FUNCTION_BLOCK fbPPPSKlimatyzatorTroxSchoolairV
  VAR_INPUT
    sKomunikat : alSTRINGKomunikat;  (* komunikat z systemu zewnętrznego *)
    intTablicaKomunikatowRozmiar : INT;  (* rozmiar tablicy danych wysyłkowych *)
    intModbusOdczytZapisZadanieRozmiar : INT;  (* rozmiar tablicy danych modbusa *)
    xTablicaKomunikatowHold : BOOL;  (* wstrzymanie komunikacji mniej ważnych komunikatów *)
    sIdInstancji : STRING;  (* parametr ID rolety np NS02L*202IBM**** *)
    sIdAplikacji : STRING;  (* parametr ID aplikacji np SO*******ECL*000 *)
    sMnemonik : STRING;  (* mnemonik właściciela - BCB* *)
    sMACAdres : STRING;  (* MAC adres sterownika *)
    sDaneZapasowe : STRING;  (* 6 znaków zapasu *)
    tCzasOpoznieniaRestartu : TIME;  (* czas opóźnienia po którym zaczynają być raportowane wartości *)
    tCzasOpoznieniaAlarmu : TIME := TIME#1m0s0ms;  (* czas opóźnienia po którym zaczynają być raportowane wartości *)
    bAdres : BYTE;
    tMinimalnyCzasRaportowania : TIME;
    tMaksymalnyCzasRaportowania : TIME;
    xAutonomizacja : BOOL;
    xAutonomizacjaSztuczna : BOOL;
  END_VAR
  VAR_IN_OUT
    arModbusOdczytCykliczny : ARRAY[1..5000] OF typModbusOdczytCykliczny;
    arModbusStatusKomunikacji : ARRAY[1..256] OF INT;
    arModbusOdczytZapisZadanie : ARRAY[1..1000] OF typModbusOdczytZapisZadanie;
    intModbusOdczytZapisZadanieZnacznikZapisu : INT;
    arTablicaKomunikatow : alARRAYTablicaKomunikatow;
    intTablicaKomunikatowZnacznikZapisu : INT;
  END_VAR
  VAR
    xPoInicjalizacji : BOOL := FALSE;  (* Inicjalizacja *)
    fbInicjalizacyjnyTimer : TON;
    tCzasInicjalizacji : TIME := TIME#30s0ms;
    xPierwszySkan : BOOL := TRUE;  (* Definicje zmiennych do odczytu wartości z modbusa *)
    intPetlaPierwszySkan : INT := 1;
    sDane : alSTRINGKomunikat;  (* Definicje do komunikacji z IZE *)
    sWyslanyKomunikat : alSTRINGKomunikat;
    sWyslanyKomunikatDummy : alSTRINGKomunikat;
    xZadanieRaportu : BOOL;
    sKomunikatPamiec : alSTRINGKomunikat;
    intPetla : INT;
    arErrorStan : ARRAY[0..10] OF INT;  (* tablica przechowująca statusy alarmowe *)
    arErrorKlasa : ARRAY[0..10] OF INT;  (* tablica przechowująca klasy danych alarmów *)
    xRaport : BOOL := FALSE;
    sTempWartoscAtrybutu : STRING;
    xOverFlow : BOOL;
    fbTimerBrakuKomunikacji : TON;  (* Kontrola komunikacji urządzenia *)
    xBrakKomunikacjiPLC : BOOL;
    xBrakKomunikacjiIZE : BOOL;
    intBlokadaWykonywaniaRozkazow : INT;  (* Parametry *)
    intBlokadaWykonywaniaRozkazowZaraportowana : INT;
    wTrybPracy : WORD;  (* 255 = Nul, 0 = Occupied, 1 = Unoccupied, 2 = Boost, 3 = Standby *)
    rTrybPracy : REAL;
    rTrybPracyZaraportowana : REAL;
    wPredkoscWentylatora : WORD;  (* High-Byte: Value, Low-Byte: 0 Auto, 1 Hand *)
    rPredkoscWentylatora : REAL;
    rPredkoscWentylatoraZaraportowana : REAL;  (* 40 = Level 1, 80 = Level 2, 120 = Level 3, 160 = Level 4, 200 = Level 5 *)
    fbPredkoscWentylatora : fbFiltrWartoscAnalogowa;
    wTrybOperacji : WORD;  (* 255 = HVAC_NUL, 0 = HVAC_AUTO, 1 = HVAC_HEAT, 2 = HVAC_MRNG_WRMUP, 3 = HVAC_COOL, 4 = HVAC_NIGHT_PURGE, 5 = HVAC_PRE_COOL, 6 = HVAC_OFF *)
    rTrybOperacji : REAL;  (* 7 = HVAC_TEST, 8 = HVAC_EMERG_HEAT, 9 = HVAC_FAN_ONLY, 10 = HVAC_FREE_COOL, 12 = HVAC_MAXHEAT, 13 = HVAC_ECONOMY, 14 = HVAC_DEHUMID *)
    rTrybOperacjiZaraportowana : REAL;
    wTemperaturaReferencyjna : WORD;  (* Unit 0.01°C *)
    rTemperaturaReferencyjna : REAL;
    rTemperaturaReferencyjnaZaraportowana : REAL;
    wTemperaturaRzeczywista : WORD;  (* Unit 0.01°C *)
    rTemperaturaRzeczywista : REAL;
    rTemperaturaRzeczywistaZaraportowana : REAL;
    fbTemperaturaRzeczywista : fbFiltrWartoscAnalogowa;
    rTemperaturaRzeczywistaPamiec : REAL;
    xBrakZmianyTemperatury : BOOL;
    fbBrakZmianyTemperaturyTimer : TON;
    xBladBrakZmianyTemperatury : BOOL;
  END_VAR

            (*			
Autor:					Artur Wyszomirski, 2019-03-08 
Prawa majątkowe: 		Solwena Sp. z o.o., 
Aktualizacje:			2019-05-16-AWy: Modyfikacja warunku na raportowanie. Dopisane: AND arModbusStatusKomunikacji[bAdres] = enumModbusStatus.KomunikacjaPrawidlowa AND xPoInicjalizacji 
						
Opis:					fb służy do komunikacji z klimatyzatorem Trox Schoolair V
				
*)


// Inicjalizacja sterownika
fbInicjalizacyjnyTimer(IN := (NOT xPoInicjalizacji AND arModbusStatusKomunikacji[bAdres] = enumModbusStatus.KomunikacjaPrawidlowa) , PT := tCzasOpoznieniaRestartu);
IF fbInicjalizacyjnyTimer.Q THEN
	rTrybPracyZaraportowana := rTrybPracy;
	rPredkoscWentylatoraZaraportowana := rPredkoscWentylatora;
	rTrybOperacji := rTrybOperacjiZaraportowana;
	rTemperaturaReferencyjnaZaraportowana := rTemperaturaReferencyjna;
	rTemperaturaRzeczywistaZaraportowana := rTemperaturaRzeczywista;
	xPoInicjalizacji := TRUE;
END_IF
//

IF xAutonomizacjaSztuczna = TRUE THEN
	xAutonomizacja := TRUE;
END_IF 

// Kontrola komunikacji
fbTimerBrakuKomunikacji(IN := arModbusStatusKomunikacji[bAdres] = enumModbusStatus.BrakKomunikacji, PT := T#60S);
IF fbTimerBrakuKomunikacji.Q THEN
	xBrakKomunikacjiPLC := TRUE;
ELSE
	xBrakKomunikacjiPLC := FALSE;
END_IF

IF xAutonomizacja THEN
	xBrakKomunikacjiIZE := TRUE;
ELSE
	xBrakKomunikacjiIZE := FALSE;
END_IF
//

IF xPierwszySkan THEN
	xPierwszySkan := FALSE;
	WHILE arModbusOdczytCykliczny[intPetlaPierwszySkan].bAdresUrzadzenia <> 0 DO
		intPetlaPierwszySkan := intPetlaPierwszySkan + 1;
	END_WHILE

	arModbusOdczytCykliczny[intPetlaPierwszySkan].bAdresUrzadzenia := bAdres;
	arModbusOdczytCykliczny[intPetlaPierwszySkan].bFunkcja := TO_BYTE(enumModbusKodyFunkcji.OdczytNRejestrowWejsciowych);
	arModbusOdczytCykliczny[intPetlaPierwszySkan].uiAdresRejestru := 17;
	arModbusOdczytCykliczny[intPetlaPierwszySkan].ltCzestotliwosc := TIME_TO_LTIME(tMinimalnyCzasRaportowania);
	arModbusOdczytCykliczny[intPetlaPierwszySkan].pZmiennaReferencyjna := ADR(wTrybPracy);
	intPetlaPierwszySkan := intPetlaPierwszySkan + 1;	
	
	arModbusOdczytCykliczny[intPetlaPierwszySkan].bAdresUrzadzenia := bAdres;
	arModbusOdczytCykliczny[intPetlaPierwszySkan].bFunkcja := TO_BYTE(enumModbusKodyFunkcji.OdczytNRejestrowWejsciowych);
	arModbusOdczytCykliczny[intPetlaPierwszySkan].uiAdresRejestru := 19;
	arModbusOdczytCykliczny[intPetlaPierwszySkan].ltCzestotliwosc := TIME_TO_LTIME(tMinimalnyCzasRaportowania);
	arModbusOdczytCykliczny[intPetlaPierwszySkan].pZmiennaReferencyjna := ADR(wTemperaturaReferencyjna);
	intPetlaPierwszySkan := intPetlaPierwszySkan + 1;		
	
	arModbusOdczytCykliczny[intPetlaPierwszySkan].bAdresUrzadzenia := bAdres;
	arModbusOdczytCykliczny[intPetlaPierwszySkan].bFunkcja := TO_BYTE(enumModbusKodyFunkcji.OdczytNRejestrowWejsciowych);
	arModbusOdczytCykliczny[intPetlaPierwszySkan].uiAdresRejestru := 21;
	arModbusOdczytCykliczny[intPetlaPierwszySkan].ltCzestotliwosc := TIME_TO_LTIME(tMinimalnyCzasRaportowania);
	arModbusOdczytCykliczny[intPetlaPierwszySkan].pZmiennaReferencyjna := ADR(wPredkoscWentylatora);
	intPetlaPierwszySkan := intPetlaPierwszySkan + 1;

	arModbusOdczytCykliczny[intPetlaPierwszySkan].bAdresUrzadzenia := bAdres;
	arModbusOdczytCykliczny[intPetlaPierwszySkan].bFunkcja := TO_BYTE(enumModbusKodyFunkcji.OdczytNRejestrowWejsciowych);
	arModbusOdczytCykliczny[intPetlaPierwszySkan].uiAdresRejestru := 22;
	arModbusOdczytCykliczny[intPetlaPierwszySkan].ltCzestotliwosc := TIME_TO_LTIME(tMinimalnyCzasRaportowania);
	arModbusOdczytCykliczny[intPetlaPierwszySkan].pZmiennaReferencyjna := ADR(wTrybOperacji);
	intPetlaPierwszySkan := intPetlaPierwszySkan + 1;

	arModbusOdczytCykliczny[intPetlaPierwszySkan].bAdresUrzadzenia := bAdres;
	arModbusOdczytCykliczny[intPetlaPierwszySkan].bFunkcja := TO_BYTE(enumModbusKodyFunkcji.OdczytNRejestrowWejsciowych);
	arModbusOdczytCykliczny[intPetlaPierwszySkan].uiAdresRejestru := 25;
	arModbusOdczytCykliczny[intPetlaPierwszySkan].ltCzestotliwosc := TIME_TO_LTIME(tMinimalnyCzasRaportowania);
	arModbusOdczytCykliczny[intPetlaPierwszySkan].pZmiennaReferencyjna := ADR(wTemperaturaRzeczywista);
	intPetlaPierwszySkan := intPetlaPierwszySkan + 1;							
END_IF

// Przeliczenie zmiennych
rTrybPracy := WORD_TO_REAL(wTrybPracy);
rPredkoscWentylatora := WORD_TO_REAL(SHR((wPredkoscWentylatora AND 16#FF00),8));
rTrybOperacji := WORD_TO_REAL(wTrybOperacji);
rTemperaturaReferencyjna := WORD_TO_REAL(wTemperaturaReferencyjna)*0.01 + 273.15;

fbTemperaturaRzeczywista(	rWartoscWejsciowa := WORD_TO_REAL(wTemperaturaRzeczywista),
							rDeadband := 0.5,
							tCzasMinimalny := tMinimalnyCzasRaportowania,
							tCzasMaksymalny := tMaksymalnyCzasRaportowania,
							rWynikMnoznik := 0.01,
							rWynikOffset := 273.15,
							rWartoscWejsciowaZaraportowana := rTemperaturaRzeczywistaZaraportowana,
							rWartoscWyjsciowa => rTemperaturaRzeczywista);
//					
						
						
// Obsluga komunikatu przychodzacego z IZE
IF sKomunikat <> sKomunikatPamiec AND xPoInicjalizacji THEN
	sKomunikatPamiec := sKomunikat;
	IF fnIDOdbiorcyMatch(sKomunikat , sIdInstancji) THEN
		sDane := '';
		// Rozkaz typu C
		IF fnKomunikatTyp(sKomunikat) = 'C' AND NOT xAutonomizacja THEN
			IF fnKomunikatDaneSzukajWartosci(sKomunikat,'BLOK=') = '0' THEN
				IF intBlokadaWykonywaniaRozkazow = 1 THEN
					intBlokadaWykonywaniaRozkazow := 0;
					xRaport := TRUE;
					ELSE	
					IF sDane <> '' THEN
					sDane := CONCAT(sDane , ';');
					END_IF
					sDane := CONCAT(sDane , 'BLOK=0');
				END_IF
			END_IF
			IF fnKomunikatDaneSzukajWartosci(sKomunikat,'BLOK=') = '1' THEN
				IF intBlokadaWykonywaniaRozkazow = 0 THEN
					intBlokadaWykonywaniaRozkazow := 1;
					xRaport := TRUE;
					ELSE
					IF sDane <> '' THEN
					sDane := CONCAT(sDane , ';');
					END_IF					
					sDane := CONCAT(sDane , 'BLOK=1');
				END_IF
			END_IF
		END_IF
				
		// Zapytanie typu Q
		IF fnKomunikatTyp(sKomunikat) = 'Q' AND arModbusStatusKomunikacji[bAdres] = enumModbusStatus.KomunikacjaPrawidlowa THEN
			IF fnKomunikatDaneSzukajWartosci(sKomunikat , 'BLOK=') = '?' OR fnKomunikatDaneSzukajWartosci(sKomunikat , 'ALL=') = '?' THEN
				fnKomunikatDaneDodaj_xOverFlow(sDane := sDane , sAtrybut := 'BLOK=' , sWartosc := INT_TO_STRING(intBlokadaWykonywaniaRozkazow) , xOverFlow := xOverFlow);	
				IF xOverFlow = TRUE THEN
					fnZapiszKomunikat(	sCalyKomunikat := '' ,
								sTypKomunikatu := 'A' ,
								sMnemonik := sMnemonik ,
								sMACAdres := sMACAdres ,
								sIDNadawcy := sIdInstancji ,
								sIDOdbiorcy := sIdAplikacji ,
								sDaneZapasowe := sDaneZapasowe ,
								sDane := sDane ,
								arTablicaKomunikatow := arTablicaKomunikatow ,
								intTablicaKomunikatowZnacznikZapisu := intTablicaKomunikatowZnacznikZapisu ,
								intTablicaKomunikatowRozmiar := intTablicaKomunikatowRozmiar ,
								sWyslanyKomunikat := sWyslanyKomunikatDummy);
					sDane := '';
				END_IF
			END_IF
			IF fnKomunikatDaneSzukajWartosci(sKomunikat , 'TRYBPRACY=') = '?' OR fnKomunikatDaneSzukajWartosci(sKomunikat , 'ALL=') = '?' THEN
				fnKomunikatDaneDodaj_xOverFlow(sDane := sDane , sAtrybut := 'TRYBPRACY=' , sWartosc := REAL_TO_STRING(rTrybPracy) , xOverFlow := xOverFlow);	
				IF xOverFlow = TRUE THEN
					fnZapiszKomunikat(	sCalyKomunikat := '' ,
								sTypKomunikatu := 'A' ,
								sMnemonik := sMnemonik ,
								sMACAdres := sMACAdres ,
								sIDNadawcy := sIdInstancji ,
								sIDOdbiorcy := sIdAplikacji ,
								sDaneZapasowe := sDaneZapasowe ,
								sDane := sDane ,
								arTablicaKomunikatow := arTablicaKomunikatow ,
								intTablicaKomunikatowZnacznikZapisu := intTablicaKomunikatowZnacznikZapisu ,
								intTablicaKomunikatowRozmiar := intTablicaKomunikatowRozmiar ,
								sWyslanyKomunikat := sWyslanyKomunikatDummy);
					sDane := '';
				END_IF
			END_IF		
			IF fnKomunikatDaneSzukajWartosci(sKomunikat , 'PREDKOSCWENT=') = '?' OR fnKomunikatDaneSzukajWartosci(sKomunikat , 'ALL=') = '?' THEN
				fnKomunikatDaneDodaj_xOverFlow(sDane := sDane , sAtrybut := 'PREDKOSCWENT=' , sWartosc := REAL_TO_STRING(rPredkoscWentylatora) , xOverFlow := xOverFlow);	
				IF xOverFlow = TRUE THEN
					fnZapiszKomunikat(	sCalyKomunikat := '' ,
								sTypKomunikatu := 'A' ,
								sMnemonik := sMnemonik ,
								sMACAdres := sMACAdres ,
								sIDNadawcy := sIdInstancji ,
								sIDOdbiorcy := sIdAplikacji ,
								sDaneZapasowe := sDaneZapasowe ,
								sDane := sDane ,
								arTablicaKomunikatow := arTablicaKomunikatow ,
								intTablicaKomunikatowZnacznikZapisu := intTablicaKomunikatowZnacznikZapisu ,
								intTablicaKomunikatowRozmiar := intTablicaKomunikatowRozmiar ,
								sWyslanyKomunikat := sWyslanyKomunikatDummy);
					sDane := '';
				END_IF
			END_IF		
			IF fnKomunikatDaneSzukajWartosci(sKomunikat , 'TEMPREF=') = '?' OR fnKomunikatDaneSzukajWartosci(sKomunikat , 'ALL=') = '?' THEN
				fnKomunikatDaneDodaj_xOverFlow(sDane := sDane , sAtrybut := 'TEMPREF=' , sWartosc := REAL_TO_STRING(rTemperaturaReferencyjna) , xOverFlow := xOverFlow);	
				IF xOverFlow = TRUE THEN
					fnZapiszKomunikat(	sCalyKomunikat := '' ,
								sTypKomunikatu := 'A' ,
								sMnemonik := sMnemonik ,
								sMACAdres := sMACAdres ,
								sIDNadawcy := sIdInstancji ,
								sIDOdbiorcy := sIdAplikacji ,
								sDaneZapasowe := sDaneZapasowe ,
								sDane := sDane ,
								arTablicaKomunikatow := arTablicaKomunikatow ,
								intTablicaKomunikatowZnacznikZapisu := intTablicaKomunikatowZnacznikZapisu ,
								intTablicaKomunikatowRozmiar := intTablicaKomunikatowRozmiar ,
								sWyslanyKomunikat := sWyslanyKomunikatDummy);
					sDane := '';
				END_IF
			END_IF		
			IF fnKomunikatDaneSzukajWartosci(sKomunikat , 'TEMPRZECZ=') = '?' OR fnKomunikatDaneSzukajWartosci(sKomunikat , 'ALL=') = '?' THEN
				fnKomunikatDaneDodaj_xOverFlow(sDane := sDane , sAtrybut := 'TEMPRZECZ=' , sWartosc := REAL_TO_STRING(rTemperaturaRzeczywista) , xOverFlow := xOverFlow);	
				IF xOverFlow = TRUE THEN
					fnZapiszKomunikat(	sCalyKomunikat := '' ,
								sTypKomunikatu := 'A' ,
								sMnemonik := sMnemonik ,
								sMACAdres := sMACAdres ,
								sIDNadawcy := sIdInstancji ,
								sIDOdbiorcy := sIdAplikacji ,
								sDaneZapasowe := sDaneZapasowe ,
								sDane := sDane ,
								arTablicaKomunikatow := arTablicaKomunikatow ,
								intTablicaKomunikatowZnacznikZapisu := intTablicaKomunikatowZnacznikZapisu ,
								intTablicaKomunikatowRozmiar := intTablicaKomunikatowRozmiar ,
								sWyslanyKomunikat := sWyslanyKomunikatDummy);
					sDane := '';
				END_IF
			END_IF		
			IF fnKomunikatDaneSzukajWartosci(sKomunikat , 'TRYBOP=') = '?' OR fnKomunikatDaneSzukajWartosci(sKomunikat , 'ALL=') = '?' THEN
				fnKomunikatDaneDodaj_xOverFlow(sDane := sDane , sAtrybut := 'TRYBOP=' , sWartosc := REAL_TO_STRING(rTrybOperacji) , xOverFlow := xOverFlow);	
				IF xOverFlow = TRUE THEN
					fnZapiszKomunikat(	sCalyKomunikat := '' ,
								sTypKomunikatu := 'A' ,
								sMnemonik := sMnemonik ,
								sMACAdres := sMACAdres ,
								sIDNadawcy := sIdInstancji ,
								sIDOdbiorcy := sIdAplikacji ,
								sDaneZapasowe := sDaneZapasowe ,
								sDane := sDane ,
								arTablicaKomunikatow := arTablicaKomunikatow ,
								intTablicaKomunikatowZnacznikZapisu := intTablicaKomunikatowZnacznikZapisu ,
								intTablicaKomunikatowRozmiar := intTablicaKomunikatowRozmiar ,
								sWyslanyKomunikat := sWyslanyKomunikatDummy);
					sDane := '';
				END_IF
			END_IF		
			// Pytanie o stany alarmów
			IF fnKomunikatDaneSzukajWartosci(sKomunikat , 'ALARM=') = '?' OR fnKomunikatDaneSzukajWartosci(sKomunikat , 'ALL=') = '?' THEN
				FOR intPetla := 1 TO 10 BY 1 DO
					// Raportowanie typu E (stanów alarmów) na zapytanie typu Q
					IF arErrorStan[intPetla] <> enumAlarmWartosc.StanNieznany THEN
						fnZapiszKomunikat(	sCalyKomunikat := '' ,
											sTypKomunikatu := 'E' ,
											sMnemonik := sMnemonik ,
											sMACAdres := sMACAdres ,
											sIDNadawcy := sIdInstancji ,
											sIDOdbiorcy := sIdAplikacji ,
											sDaneZapasowe := sDaneZapasowe ,
											sDane := fnKomunikatDaneErrorRetry(xAktywny := arErrorStan[intPetla] = enumAlarmWartosc.StanAlarmowy , intKlasa := arErrorKlasa[intPetla] , intNumer := intPetla),
											arTablicaKomunikatow := arTablicaKomunikatow ,
											intTablicaKomunikatowZnacznikZapisu := intTablicaKomunikatowZnacznikZapisu ,
											intTablicaKomunikatowRozmiar := intTablicaKomunikatowRozmiar ,
											sWyslanyKomunikat := sWyslanyKomunikatDummy);
					END_IF
				END_FOR
			END_IF
		END_IF		
		// Raportowanie typu A na zapytanie Q
		IF sDane <> '' THEN
			fnZapiszKomunikat(	sCalyKomunikat := '' ,
								sTypKomunikatu := 'A' ,
								sMnemonik := sMnemonik ,
								sMACAdres := sMACAdres ,
								sIDNadawcy := sIdInstancji ,
								sIDOdbiorcy := sIdAplikacji ,
								sDaneZapasowe := sDaneZapasowe ,
								sDane := sDane ,
								arTablicaKomunikatow := arTablicaKomunikatow ,
								intTablicaKomunikatowZnacznikZapisu := intTablicaKomunikatowZnacznikZapisu ,
								intTablicaKomunikatowRozmiar := intTablicaKomunikatowRozmiar ,
								sWyslanyKomunikat := sWyslanyKomunikatDummy);
		END_IF
	END_IF
END_IF

// Raportowanie typu M do IZE wartosci odczytanych z Modbusa	
IF 	(intBlokadaWykonywaniaRozkazow <> intBlokadaWykonywaniaRozkazowZaraportowana OR rTrybPracy <> rTrybPracyZaraportowana OR rPredkoscWentylatora <> rPredkoscWentylatoraZaraportowana OR
	rTemperaturaReferencyjna <> rTemperaturaReferencyjnaZaraportowana OR rTemperaturaRzeczywista <> rTemperaturaRzeczywistaZaraportowana OR rTrybOperacji <> rTrybOperacjiZaraportowana) AND 
	arModbusStatusKomunikacji[bAdres] = enumModbusStatus.KomunikacjaPrawidlowa AND xPoInicjalizacji THEN
	xRaport := TRUE;
END_IF

IF xRaport THEN
	sDane := '';
	xRaport := FALSE;
	IF intBlokadaWykonywaniaRozkazow <> intBlokadaWykonywaniaRozkazowZaraportowana THEN 
		intBlokadaWykonywaniaRozkazowZaraportowana := intBlokadaWykonywaniaRozkazow;
		fnKomunikatDaneDodaj_xOverFlow(sDane := sDane , sAtrybut := 'BLOK=' , sWartosc := INT_TO_STRING(intBlokadaWykonywaniaRozkazow) , xOverFlow := xOverFlow);	
	END_IF	
	IF xOverFlow = TRUE THEN
		fnZapiszKomunikat(	sCalyKomunikat := '' ,
					sTypKomunikatu := 'M' ,
					sMnemonik := sMnemonik ,
					sMACAdres := sMACAdres ,
					sIDNadawcy := sIdInstancji ,
					sIDOdbiorcy := sIdAplikacji ,
					sDaneZapasowe := sDaneZapasowe ,
					sDane := sDane ,
					arTablicaKomunikatow := arTablicaKomunikatow ,
					intTablicaKomunikatowZnacznikZapisu := intTablicaKomunikatowZnacznikZapisu ,
					intTablicaKomunikatowRozmiar := intTablicaKomunikatowRozmiar ,
					sWyslanyKomunikat := sWyslanyKomunikatDummy);
		sDane := '';
	END_IF
	// Tryb pracy
	IF rTrybPracy <> rTrybPracyZaraportowana THEN
		rTrybPracyZaraportowana := rTrybPracy;
		fnKomunikatDaneDodaj_xOverFlow(sDane := sDane , sAtrybut := 'TRYBPRACY=' , sWartosc := REAL_TO_STRING(rTrybPracy) , xOverFlow := xOverFlow);	
		IF xOverFlow = TRUE THEN
			fnZapiszKomunikat(	sCalyKomunikat := '' ,
						sTypKomunikatu := 'M' ,
						sMnemonik := sMnemonik ,
						sMACAdres := sMACAdres ,
						sIDNadawcy := sIdInstancji ,
						sIDOdbiorcy := sIdAplikacji ,
						sDaneZapasowe := sDaneZapasowe ,
						sDane := sDane ,
						arTablicaKomunikatow := arTablicaKomunikatow ,
						intTablicaKomunikatowZnacznikZapisu := intTablicaKomunikatowZnacznikZapisu ,
						intTablicaKomunikatowRozmiar := intTablicaKomunikatowRozmiar ,
						sWyslanyKomunikat := sWyslanyKomunikatDummy);
			sDane := '';
		END_IF	
	END_IF
	// Prędkość wentylatora
	IF rPredkoscWentylatora <> rPredkoscWentylatoraZaraportowana THEN
		rPredkoscWentylatoraZaraportowana := rPredkoscWentylatora;
		fnKomunikatDaneDodaj_xOverFlow(sDane := sDane , sAtrybut := 'PREDKOSCWENT=' , sWartosc := REAL_TO_STRING(rPredkoscWentylatora) , xOverFlow := xOverFlow);	
		IF xOverFlow = TRUE THEN
			fnZapiszKomunikat(	sCalyKomunikat := '' ,
						sTypKomunikatu := 'M' ,
						sMnemonik := sMnemonik ,
						sMACAdres := sMACAdres ,
						sIDNadawcy := sIdInstancji ,
						sIDOdbiorcy := sIdAplikacji ,
						sDaneZapasowe := sDaneZapasowe ,
						sDane := sDane ,
						arTablicaKomunikatow := arTablicaKomunikatow ,
						intTablicaKomunikatowZnacznikZapisu := intTablicaKomunikatowZnacznikZapisu ,
						intTablicaKomunikatowRozmiar := intTablicaKomunikatowRozmiar ,
						sWyslanyKomunikat := sWyslanyKomunikatDummy);
			sDane := '';
		END_IF	
	END_IF
	// Temperatura referencyjna
	IF rTemperaturaReferencyjna <> rTemperaturaReferencyjnaZaraportowana THEN
		rTemperaturaReferencyjnaZaraportowana := rTemperaturaReferencyjna;
		fnKomunikatDaneDodaj_xOverFlow(sDane := sDane , sAtrybut := 'TEMPREF=' , sWartosc := REAL_TO_STRING(rTemperaturaReferencyjna) , xOverFlow := xOverFlow);	
		IF xOverFlow = TRUE THEN
			fnZapiszKomunikat(	sCalyKomunikat := '' ,
						sTypKomunikatu := 'M' ,
						sMnemonik := sMnemonik ,
						sMACAdres := sMACAdres ,
						sIDNadawcy := sIdInstancji ,
						sIDOdbiorcy := sIdAplikacji ,
						sDaneZapasowe := sDaneZapasowe ,
						sDane := sDane ,
						arTablicaKomunikatow := arTablicaKomunikatow ,
						intTablicaKomunikatowZnacznikZapisu := intTablicaKomunikatowZnacznikZapisu ,
						intTablicaKomunikatowRozmiar := intTablicaKomunikatowRozmiar ,
						sWyslanyKomunikat := sWyslanyKomunikatDummy);
			sDane := '';
		END_IF	
	END_IF
	// Temperatura rzeczywista
	IF rTemperaturaRzeczywista <> rTemperaturaRzeczywistaZaraportowana THEN
		rTemperaturaRzeczywistaZaraportowana := rTemperaturaRzeczywista;
		fnKomunikatDaneDodaj_xOverFlow(sDane := sDane , sAtrybut := 'TEMPRZECZ=' , sWartosc := REAL_TO_STRING(rTemperaturaRzeczywista) , xOverFlow := xOverFlow);	
		IF xOverFlow = TRUE THEN
			fnZapiszKomunikat(	sCalyKomunikat := '' ,
						sTypKomunikatu := 'M' ,
						sMnemonik := sMnemonik ,
						sMACAdres := sMACAdres ,
						sIDNadawcy := sIdInstancji ,
						sIDOdbiorcy := sIdAplikacji ,
						sDaneZapasowe := sDaneZapasowe ,
						sDane := sDane ,
						arTablicaKomunikatow := arTablicaKomunikatow ,
						intTablicaKomunikatowZnacznikZapisu := intTablicaKomunikatowZnacznikZapisu ,
						intTablicaKomunikatowRozmiar := intTablicaKomunikatowRozmiar ,
						sWyslanyKomunikat := sWyslanyKomunikatDummy);
			sDane := '';
		END_IF	
	END_IF
	// Temperatura referencyjna trybu manulnego
	IF rTrybOperacji <> rTrybOperacjiZaraportowana THEN
		rTrybOperacjiZaraportowana := rTrybOperacji;
		fnKomunikatDaneDodaj_xOverFlow(sDane := sDane , sAtrybut := 'TRYBOP=' , sWartosc := REAL_TO_STRING(rTrybOperacji) , xOverFlow := xOverFlow);	
		IF xOverFlow = TRUE THEN
			fnZapiszKomunikat(	sCalyKomunikat := '' ,
						sTypKomunikatu := 'M' ,
						sMnemonik := sMnemonik ,
						sMACAdres := sMACAdres ,
						sIDNadawcy := sIdInstancji ,
						sIDOdbiorcy := sIdAplikacji ,
						sDaneZapasowe := sDaneZapasowe ,
						sDane := sDane ,
						arTablicaKomunikatow := arTablicaKomunikatow ,
						intTablicaKomunikatowZnacznikZapisu := intTablicaKomunikatowZnacznikZapisu ,
						intTablicaKomunikatowRozmiar := intTablicaKomunikatowRozmiar ,
						sWyslanyKomunikat := sWyslanyKomunikatDummy);
			sDane := '';
		END_IF	
	END_IF
	IF sDane <> '' AND xPoInicjalizacji THEN
	fnZapiszKomunikat(	sCalyKomunikat := '' ,
						sTypKomunikatu := 'M' ,
						sMnemonik := sMnemonik ,
						sMACAdres := sMACAdres ,
						sIDNadawcy := sIdInstancji ,
						sIDOdbiorcy := sIdAplikacji ,
						sDaneZapasowe := sDaneZapasowe ,
						sDane := sDane ,
						arTablicaKomunikatow := arTablicaKomunikatow ,
						intTablicaKomunikatowZnacznikZapisu := intTablicaKomunikatowZnacznikZapisu ,
						intTablicaKomunikatowRozmiar := intTablicaKomunikatowRozmiar ,
						sWyslanyKomunikat := sWyslanyKomunikat);
	END_IF
END_IF

// Sprawdzanie czy pomiar temperatury działa (odczyt jest niepoprawny, jeśli nie zmienił wartości w przeciągu doby)
IF rTemperaturaRzeczywistaPamiec = rTemperaturaRzeczywista THEN
	xBrakZmianyTemperatury := TRUE;
ELSE
	xBrakZmianyTemperatury := FALSE;	
END_IF
fbBrakZmianyTemperaturyTimer(IN := xBrakZmianyTemperatury, PT := T#12H);
rTemperaturaRzeczywistaPamiec := rTemperaturaRzeczywista;
IF fbBrakZmianyTemperaturyTimer.Q THEN
	xBladBrakZmianyTemperatury := TRUE;
ELSE
	xBladBrakZmianyTemperatury := FALSE;
END_IF

// Alarm braku komunikacji MODBUS 
IF arErrorStan[enumPPPSKlimatyzatorTroxSchoolairVError.BrakKomunikacji] <> enumAlarmWartosc.StanAlarmowy AND arModbusStatusKomunikacji[bAdres] = enumModbusStatus.BrakKomunikacji THEN
	arErrorStan[enumPPPSKlimatyzatorTroxSchoolairVError.BrakKomunikacji] := enumAlarmWartosc.StanAlarmowy;
	arErrorKlasa[enumPPPSKlimatyzatorTroxSchoolairVError.BrakKomunikacji] := enumPPPSKlimatyzatorTroxSchoolairVErrorKlasa.BrakKomunikacji;
	IF xPoInicjalizacji THEN
		fnZapiszKomunikat(	sCalyKomunikat := '' ,
							sTypKomunikatu := 'E' ,
							sMnemonik := sMnemonik ,
							sMACAdres := sMACAdres ,
							sIDNadawcy := sIdInstancji ,
							sIDOdbiorcy := sIdAplikacji ,
							sDaneZapasowe := sDaneZapasowe ,
							sDane := fnKomunikatDaneError(xAktywny := TRUE , intKlasa := enumPPPSKlimatyzatorTroxSchoolairVErrorKlasa.BrakKomunikacji , intNumer := enumPPPSKlimatyzatorTroxSchoolairVError.BrakKomunikacji),
							arTablicaKomunikatow := arTablicaKomunikatow ,
							intTablicaKomunikatowZnacznikZapisu := intTablicaKomunikatowZnacznikZapisu ,
							intTablicaKomunikatowRozmiar := intTablicaKomunikatowRozmiar ,
							sWyslanyKomunikat := sWyslanyKomunikatDummy);
	END_IF
END_IF
IF arErrorStan[enumPPPSKlimatyzatorTroxSchoolairVError.BrakKomunikacji] <> enumAlarmWartosc.StanNormalny AND arModbusStatusKomunikacji[bAdres] = enumModbusStatus.KomunikacjaPrawidlowa THEN
	arErrorStan[enumPPPSKlimatyzatorTroxSchoolairVError.BrakKomunikacji] := enumAlarmWartosc.StanNormalny;
	arErrorKlasa[enumPPPSKlimatyzatorTroxSchoolairVError.BrakKomunikacji] := enumPPPSKlimatyzatorTroxSchoolairVErrorKlasa.BrakKomunikacji;
	IF xPoInicjalizacji THEN
		fnZapiszKomunikat(	sCalyKomunikat := '' ,
							sTypKomunikatu := 'E' ,
							sMnemonik := sMnemonik ,
							sMACAdres := sMACAdres ,
							sIDNadawcy := sIdInstancji ,
							sIDOdbiorcy := sIdAplikacji ,
							sDaneZapasowe := sDaneZapasowe ,
							sDane := fnKomunikatDaneError(xAktywny := FALSE , intKlasa := enumPPPSKlimatyzatorTroxSchoolairVErrorKlasa.BrakKomunikacji , intNumer := enumPPPSKlimatyzatorTroxSchoolairVError.BrakKomunikacji),
							arTablicaKomunikatow := arTablicaKomunikatow ,
							intTablicaKomunikatowZnacznikZapisu := intTablicaKomunikatowZnacznikZapisu ,
							intTablicaKomunikatowRozmiar := intTablicaKomunikatowRozmiar ,
							sWyslanyKomunikat := sWyslanyKomunikatDummy);
	END_IF
END_IF

// Alarm czujnika temperatury
IF arErrorStan[enumPPPSKlimatyzatorTroxSchoolairVError.AlarmCzujnika] <> enumAlarmWartosc.StanAlarmowy AND xBladBrakZmianyTemperatury AND arModbusStatusKomunikacji[bAdres] = enumModbusStatus.KomunikacjaPrawidlowa THEN
	arErrorStan[enumPPPSKlimatyzatorTroxSchoolairVError.AlarmCzujnika] := enumAlarmWartosc.StanAlarmowy;
	arErrorKlasa[enumPPPSKlimatyzatorTroxSchoolairVError.AlarmCzujnika] := enumPPPSKlimatyzatorTroxSchoolairVErrorKlasa.AlarmCzujnika;
	IF xPoInicjalizacji THEN
		fnZapiszKomunikat(	sCalyKomunikat := '' ,
							sTypKomunikatu := 'E' ,
							sMnemonik := sMnemonik ,
							sMACAdres := sMACAdres ,
							sIDNadawcy := sIdInstancji ,
							sIDOdbiorcy := sIdAplikacji ,
							sDaneZapasowe := sDaneZapasowe ,
							sDane := fnKomunikatDaneError(xAktywny := TRUE , intKlasa := enumPPPSKlimatyzatorTroxSchoolairVErrorKlasa.AlarmCzujnika , intNumer := enumPPPSKlimatyzatorTroxSchoolairVError.AlarmCzujnika),
							arTablicaKomunikatow := arTablicaKomunikatow ,
							intTablicaKomunikatowZnacznikZapisu := intTablicaKomunikatowZnacznikZapisu ,
							intTablicaKomunikatowRozmiar := intTablicaKomunikatowRozmiar ,
							sWyslanyKomunikat := sWyslanyKomunikatDummy);
	END_IF
END_IF
IF arErrorStan[enumPPPSKlimatyzatorTroxSchoolairVError.AlarmCzujnika] <> enumAlarmWartosc.StanNormalny AND NOT xBladBrakZmianyTemperatury AND arModbusStatusKomunikacji[bAdres] = enumModbusStatus.KomunikacjaPrawidlowa THEN
	arErrorStan[enumPPPSKlimatyzatorTroxSchoolairVError.AlarmCzujnika] := enumAlarmWartosc.StanNormalny;
	arErrorKlasa[enumPPPSKlimatyzatorTroxSchoolairVError.AlarmCzujnika] := enumPPPSKlimatyzatorTroxSchoolairVErrorKlasa.AlarmCzujnika;
	IF xPoInicjalizacji THEN
		fnZapiszKomunikat(	sCalyKomunikat := '' ,
							sTypKomunikatu := 'E' ,
							sMnemonik := sMnemonik ,
							sMACAdres := sMACAdres ,
							sIDNadawcy := sIdInstancji ,
							sIDOdbiorcy := sIdAplikacji ,
							sDaneZapasowe := sDaneZapasowe ,
							sDane := fnKomunikatDaneError(xAktywny := FALSE , intKlasa := enumPPPSKlimatyzatorTroxSchoolairVErrorKlasa.AlarmCzujnika , intNumer := enumPPPSKlimatyzatorTroxSchoolairVError.AlarmCzujnika),
							arTablicaKomunikatow := arTablicaKomunikatow ,
							intTablicaKomunikatowZnacznikZapisu := intTablicaKomunikatowZnacznikZapisu ,
							intTablicaKomunikatowRozmiar := intTablicaKomunikatowRozmiar ,
							sWyslanyKomunikat := sWyslanyKomunikatDummy);
	END_IF
END_IF

          
END_FUNCTION_BLOCK

FUNCTION_BLOCK fbPPPSLicznikCieplaMultical403
  VAR_INPUT
    sKomunikat : alSTRINGKomunikat;  (* komunikat z systemu zewnętrznego *)
    intTablicaKomunikatowRozmiar : INT;  (* rozmiar tablicy danych wysyłkowych *)
    intModbusOdczytZapisZadanieRozmiar : INT;  (* rozmiar tablicy danych modbusa *)
    xTablicaKomunikatowHold : BOOL;  (* wstrzymanie komunikacji mniej ważnych komunikatów *)
    sIdInstancji : STRING;  (* parametr ID rolety np NS02L*202IBM**** *)
    sIdAplikacji : STRING;  (* parametr ID aplikacji np SO*******ECL*000 *)
    sMnemonik : STRING;  (* mnemonik właściciela - BCB* *)
    sMACAdres : STRING;  (* MAC adres sterownika *)
    sDaneZapasowe : STRING;  (* 6 znaków zapasu *)
    tCzasOpoznieniaRestartu : TIME;  (* czas opóźnienia po którym zaczynają być raportowane wartości *)
    tCzasOpoznieniaAlarmu : TIME := TIME#1m0s0ms;  (* czas opóźnienia po którym zaczynają być raportowane wartości *)
    bAdres : BYTE;
    tMinimalnyCzasRaportowania : TIME;
    tMaksymalnyCzasRaportowania : TIME;
    xAutonomizacja : BOOL;
    xAutonomizacjaSztuczna : BOOL;
  END_VAR
  VAR_IN_OUT
    arModbusOdczytCykliczny : ARRAY[1..5000] OF typModbusOdczytCykliczny;
    arModbusStatusKomunikacji : ARRAY[1..256] OF INT;
    arTablicaKomunikatow : alARRAYTablicaKomunikatow;
    intTablicaKomunikatowZnacznikZapisu : INT;
  END_VAR
  VAR
    xPoInicjalizacji : BOOL := FALSE;  (* Inicjalizacja *)
    fbInicjalizacyjnyTimer : TON;
    tCzasInicjalizacji : TIME := TIME#30s0ms;
    xPierwszySkan : BOOL := TRUE;  (* Definicje zmiennych do odczytu wartości z modbusa *)
    intPetlaPierwszySkan : INT := 1;
    sDane : alSTRINGKomunikat;  (* Definicje do komunikacji z IZE *)
    sWyslanyKomunikat : alSTRINGKomunikat;
    sWyslanyKomunikatDummy : alSTRINGKomunikat;
    xZadanieRaportu : BOOL;
    sKomunikatPamiec : alSTRINGKomunikat;
    intPetla : INT;
    arErrorStan : ARRAY[0..10] OF INT;  (* tablica przechowująca statusy alarmowe *)
    arErrorKlasa : ARRAY[0..10] OF INT;  (* tablica przechowująca klasy danych alarmów *)
    xRaport : BOOL := FALSE;
    sTempWartoscAtrybutu : STRING;
    xOverFlow : BOOL;
    fbTimerBrakuKomunikacji : TON;  (* Kontrola komunikacji urządzenia *)
    xBrakKomunikacjiPLC : BOOL;
    xBrakKomunikacjiIZE : BOOL;
    wEnergiaCieplna_Lo : WORD;  (* Całkowita energia cieplna *)
    wEnergiaCieplna_Hi : WORD;
    rEnergiaCieplna : REAL;
    fbEnergiaCieplna : fbFiltrWartoscAnalogowa;
    rEnergiaCieplnaZaraportowana : REAL;
    wEnergiaCieplnaJednostka : WORD;  (* Jednostka energii cieplnej *)
    wPrzeplyw_Lo : WORD;  (* Aktualna wartość przepływu *)
    wPrzeplyw_Hi : WORD;
    rPrzeplyw : REAL;
    fbPrzeplyw : fbFiltrWartoscAnalogowa;
    rPrzeplywZaraportowana : REAL;
    wPrzeplywJednostka : WORD;  (* Jednostka przepływu *)
    rPrzeplywPamiec : REAL;  (* Wartosc przechowywana w pamieci w celu porównania z wartością aktualną *)
    xBrakZmianyPrzeplywu : BOOL;  (* Flaga informująca o braku zmiany przepływu w czasie *)
    fbBrakZmianyPrzeplywuTimer : TON;
    xBladBrakZmianyPrzeplywu : BOOL;  (* Flaga informująca o braku przeplywu przez czas 12h - podstawa wygenerowania alarmu *)
    wObjetosc_Lo : WORD;  (* Objętość medium, które przepłynęło przez licznik *)
    wObjetosc_Hi : WORD;
    rObjetosc : REAL;
    fbObjetosc : fbFiltrWartoscAnalogowa;
    rObjetoscZaraportowana : REAL;
    wObjetoscJednostka : WORD;  (* Jednostka wolumenu *)
    wMoc_Hi : WORD;  (* Aktualna moc cieplna płynąca przez licznik *)
    wMoc_Lo : WORD;
    rMoc : REAL;
    fbMoc : fbFiltrWartoscAnalogowa;
    rMocZaraportowana : REAL;
    wMocJednostka : WORD;  (* Jednostka mocy *)
    wTemperaturaZasilania_Lo : WORD;  (* Temp czynnika na wejściu licznika *)
    wTemperaturaZasilania_Hi : WORD;
    rTemperaturaZasilania : REAL;
    fbTemperaturaZasilania : fbFiltrWartoscAnalogowa;
    rTemperaturaZasilaniaZaraportowana : REAL;
    rTemperaturaZasilaniaPamiec : REAL;  (* Wartosc przechowywana w pamieci w celu porównania z wartością aktualną *)
    xBrakZmianyTemperaturyZasilania : BOOL;  (* Flaga informująca o braku zmiany przepływu w czasie *)
    fbBrakZmianyTemperaturyZasilaniaTimer : TON;
    xBladBrakZmianyTemperaturyZasilania : BOOL;  (* Flaga informująca o braku przeplywu przez czas 12h - podstawa wygenerowania alarmu *)
    wTemperaturaPowrotu_Lo : WORD;  (* Temp czynnika na wyjściu licznika *)
    wTemperaturaPowrotu_Hi : WORD;
    rTemperaturaPowrotu : REAL;
    fbTemperaturaPowrotu : fbFiltrWartoscAnalogowa;
    rTemperaturaPowrotuZaraportowana : REAL;
    rTemperaturaPowrotuPamiec : REAL;  (* Wartosc przechowywana w pamieci w celu porównania z wartością aktualną *)
    xBrakZmianyTemperaturyPowrotu : BOOL;  (* Flaga informująca o braku zmiany przepływu w czasie *)
    fbBrakZmianyTemperaturyPowrotuTimer : TON;
    xBladBrakZmianyTemperaturyPowrotu : BOOL;  (* Flaga informująca o braku przeplywu przez czas 12h - podstawa wygenerowania alarmu *)
  END_VAR

            (*			
Autor:					Artur Wyszomirski, 2019-08-07 
Prawa majątkowe: 		Solwena Sp. z o.o., 
Aktualizacje:			2019-08-28-AWy: Zmiana adresów rejestrów (przesunięcie -1). Zmiana poszczególnych parametrów przy przeliczaniu zmiennych.
						2019-08-29-AWy: Usunięcie buga z raporotwania mocy.
					
Opis:					Komunikacji z licznikami ciepła Multical 403
		
*)

// Inicjalizacja sterownika
fbInicjalizacyjnyTimer(IN := (NOT xPoInicjalizacji AND arModbusStatusKomunikacji[bAdres] = enumModbusStatus.KomunikacjaPrawidlowa), PT := tCzasOpoznieniaRestartu);
IF fbInicjalizacyjnyTimer.Q THEN
	rPrzeplywZaraportowana := rPrzeplyw;
	rMocZaraportowana := rMoc;
	rEnergiaCieplnaZaraportowana := rEnergiaCieplna;
	rObjetoscZaraportowana := rObjetosc;
	rTemperaturaZasilaniaZaraportowana := rTemperaturaZasilania;
	rTemperaturaPowrotuZaraportowana := rTemperaturaPowrotu;
	xPoInicjalizacji := TRUE;
END_IF

// Włącz autonomizację jeśli sterownik jest w stanie inicjalizacji lub nastąpiło wymuszenie autonomizacji
IF NOT xPoInicjalizacji OR xAutonomizacjaSztuczna = TRUE THEN
	xAutonomizacja := TRUE;
END_IF 

// Kontrola komunikacji
fbTimerBrakuKomunikacji(IN := arModbusStatusKomunikacji[bAdres] = enumModbusStatus.BrakKomunikacji, PT := T#60S);
IF fbTimerBrakuKomunikacji.Q THEN
	xBrakKomunikacjiPLC := TRUE;
ELSE
	xBrakKomunikacjiPLC := FALSE;
END_IF

IF xAutonomizacja THEN
	xBrakKomunikacjiIZE := TRUE;
ELSE
	xBrakKomunikacjiIZE := FALSE;
END_IF

// Deklaracja rejestrów Modbusa
IF xPierwszySkan THEN
	xPierwszySkan := FALSE;
	WHILE arModbusOdczytCykliczny[intPetlaPierwszySkan].bAdresUrzadzenia <> 0 DO
		intPetlaPierwszySkan := intPetlaPierwszySkan + 1;
	END_WHILE
	arModbusOdczytCykliczny[intPetlaPierwszySkan].bAdresUrzadzenia := bAdres;
	arModbusOdczytCykliczny[intPetlaPierwszySkan].bFunkcja := TO_BYTE(enumModbusKodyFunkcji.OdczytNRejestrow);
	arModbusOdczytCykliczny[intPetlaPierwszySkan].uiAdresRejestru := 20;
	arModbusOdczytCykliczny[intPetlaPierwszySkan].ltCzestotliwosc := TIME_TO_LTIME(tMinimalnyCzasRaportowania);
	arModbusOdczytCykliczny[intPetlaPierwszySkan].pZmiennaReferencyjna := ADR(wEnergiaCieplna_Hi);
	intPetlaPierwszySkan := intPetlaPierwszySkan + 1;	
	
	arModbusOdczytCykliczny[intPetlaPierwszySkan].bAdresUrzadzenia := bAdres;
	arModbusOdczytCykliczny[intPetlaPierwszySkan].bFunkcja := TO_BYTE(enumModbusKodyFunkcji.OdczytNRejestrow);
	arModbusOdczytCykliczny[intPetlaPierwszySkan].uiAdresRejestru := 21;
	arModbusOdczytCykliczny[intPetlaPierwszySkan].ltCzestotliwosc := TIME_TO_LTIME(tMinimalnyCzasRaportowania);
	arModbusOdczytCykliczny[intPetlaPierwszySkan].pZmiennaReferencyjna := ADR(wEnergiaCieplna_Lo);
	intPetlaPierwszySkan := intPetlaPierwszySkan + 1;	
	
	arModbusOdczytCykliczny[intPetlaPierwszySkan].bAdresUrzadzenia := bAdres;
	arModbusOdczytCykliczny[intPetlaPierwszySkan].bFunkcja := TO_BYTE(enumModbusKodyFunkcji.OdczytNRejestrow);
	arModbusOdczytCykliczny[intPetlaPierwszySkan].uiAdresRejestru := 0;
	arModbusOdczytCykliczny[intPetlaPierwszySkan].ltCzestotliwosc := TIME_TO_LTIME(tMinimalnyCzasRaportowania);
	arModbusOdczytCykliczny[intPetlaPierwszySkan].pZmiennaReferencyjna := ADR(wPrzeplyw_Hi);
	intPetlaPierwszySkan := intPetlaPierwszySkan + 1;

	arModbusOdczytCykliczny[intPetlaPierwszySkan].bAdresUrzadzenia := bAdres;
	arModbusOdczytCykliczny[intPetlaPierwszySkan].bFunkcja := TO_BYTE(enumModbusKodyFunkcji.OdczytNRejestrow);
	arModbusOdczytCykliczny[intPetlaPierwszySkan].uiAdresRejestru := 1;
	arModbusOdczytCykliczny[intPetlaPierwszySkan].ltCzestotliwosc := TIME_TO_LTIME(tMinimalnyCzasRaportowania);
	arModbusOdczytCykliczny[intPetlaPierwszySkan].pZmiennaReferencyjna := ADR(wPrzeplyw_Lo);
	intPetlaPierwszySkan := intPetlaPierwszySkan + 1;
	
	arModbusOdczytCykliczny[intPetlaPierwszySkan].bAdresUrzadzenia := bAdres;
	arModbusOdczytCykliczny[intPetlaPierwszySkan].bFunkcja := TO_BYTE(enumModbusKodyFunkcji.OdczytNRejestrow);
	arModbusOdczytCykliczny[intPetlaPierwszySkan].uiAdresRejestru := 52;
	arModbusOdczytCykliczny[intPetlaPierwszySkan].ltCzestotliwosc := TIME_TO_LTIME(tMinimalnyCzasRaportowania);
	arModbusOdczytCykliczny[intPetlaPierwszySkan].pZmiennaReferencyjna := ADR(wObjetosc_Hi);
	intPetlaPierwszySkan := intPetlaPierwszySkan + 1;
	
	arModbusOdczytCykliczny[intPetlaPierwszySkan].bAdresUrzadzenia := bAdres;
	arModbusOdczytCykliczny[intPetlaPierwszySkan].bFunkcja := TO_BYTE(enumModbusKodyFunkcji.OdczytNRejestrow);
	arModbusOdczytCykliczny[intPetlaPierwszySkan].uiAdresRejestru := 53;
	arModbusOdczytCykliczny[intPetlaPierwszySkan].ltCzestotliwosc := TIME_TO_LTIME(tMinimalnyCzasRaportowania);
	arModbusOdczytCykliczny[intPetlaPierwszySkan].pZmiennaReferencyjna := ADR(wObjetosc_Lo);
	intPetlaPierwszySkan := intPetlaPierwszySkan + 1;
	
	arModbusOdczytCykliczny[intPetlaPierwszySkan].bAdresUrzadzenia := bAdres;
	arModbusOdczytCykliczny[intPetlaPierwszySkan].bFunkcja := TO_BYTE(enumModbusKodyFunkcji.OdczytNRejestrow);
	arModbusOdczytCykliczny[intPetlaPierwszySkan].uiAdresRejestru := 4;
	arModbusOdczytCykliczny[intPetlaPierwszySkan].ltCzestotliwosc := TIME_TO_LTIME(tMinimalnyCzasRaportowania);
	arModbusOdczytCykliczny[intPetlaPierwszySkan].pZmiennaReferencyjna := ADR(wMoc_Hi);
	intPetlaPierwszySkan := intPetlaPierwszySkan + 1;	
	
	arModbusOdczytCykliczny[intPetlaPierwszySkan].bAdresUrzadzenia := bAdres;
	arModbusOdczytCykliczny[intPetlaPierwszySkan].bFunkcja := TO_BYTE(enumModbusKodyFunkcji.OdczytNRejestrow);
	arModbusOdczytCykliczny[intPetlaPierwszySkan].uiAdresRejestru := 5;
	arModbusOdczytCykliczny[intPetlaPierwszySkan].ltCzestotliwosc := TIME_TO_LTIME(tMinimalnyCzasRaportowania);
	arModbusOdczytCykliczny[intPetlaPierwszySkan].pZmiennaReferencyjna := ADR(wMoc_Lo);
	intPetlaPierwszySkan := intPetlaPierwszySkan + 1;
	
	arModbusOdczytCykliczny[intPetlaPierwszySkan].bAdresUrzadzenia := bAdres;
	arModbusOdczytCykliczny[intPetlaPierwszySkan].bFunkcja := TO_BYTE(enumModbusKodyFunkcji.OdczytNRejestrow);
	arModbusOdczytCykliczny[intPetlaPierwszySkan].uiAdresRejestru := 6;
	arModbusOdczytCykliczny[intPetlaPierwszySkan].ltCzestotliwosc := TIME_TO_LTIME(tMinimalnyCzasRaportowania);
	arModbusOdczytCykliczny[intPetlaPierwszySkan].pZmiennaReferencyjna := ADR(wTemperaturaZasilania_Hi);
	intPetlaPierwszySkan := intPetlaPierwszySkan + 1;	
	
	arModbusOdczytCykliczny[intPetlaPierwszySkan].bAdresUrzadzenia := bAdres;
	arModbusOdczytCykliczny[intPetlaPierwszySkan].bFunkcja := TO_BYTE(enumModbusKodyFunkcji.OdczytNRejestrow);
	arModbusOdczytCykliczny[intPetlaPierwszySkan].uiAdresRejestru := 7;
	arModbusOdczytCykliczny[intPetlaPierwszySkan].ltCzestotliwosc := TIME_TO_LTIME(tMinimalnyCzasRaportowania);
	arModbusOdczytCykliczny[intPetlaPierwszySkan].pZmiennaReferencyjna := ADR(wTemperaturaZasilania_Lo);
	intPetlaPierwszySkan := intPetlaPierwszySkan + 1;
	
	arModbusOdczytCykliczny[intPetlaPierwszySkan].bAdresUrzadzenia := bAdres;
	arModbusOdczytCykliczny[intPetlaPierwszySkan].bFunkcja := TO_BYTE(enumModbusKodyFunkcji.OdczytNRejestrow);
	arModbusOdczytCykliczny[intPetlaPierwszySkan].uiAdresRejestru := 8;
	arModbusOdczytCykliczny[intPetlaPierwszySkan].ltCzestotliwosc := TIME_TO_LTIME(tMinimalnyCzasRaportowania);
	arModbusOdczytCykliczny[intPetlaPierwszySkan].pZmiennaReferencyjna := ADR(wTemperaturaPowrotu_Hi);
	intPetlaPierwszySkan := intPetlaPierwszySkan + 1;	
	
	arModbusOdczytCykliczny[intPetlaPierwszySkan].bAdresUrzadzenia := bAdres;
	arModbusOdczytCykliczny[intPetlaPierwszySkan].bFunkcja := TO_BYTE(enumModbusKodyFunkcji.OdczytNRejestrow);
	arModbusOdczytCykliczny[intPetlaPierwszySkan].uiAdresRejestru := 9;
	arModbusOdczytCykliczny[intPetlaPierwszySkan].ltCzestotliwosc := TIME_TO_LTIME(tMinimalnyCzasRaportowania);
	arModbusOdczytCykliczny[intPetlaPierwszySkan].pZmiennaReferencyjna := ADR(wTemperaturaPowrotu_Lo);
	intPetlaPierwszySkan := intPetlaPierwszySkan + 1;
	
	arModbusOdczytCykliczny[intPetlaPierwszySkan].bAdresUrzadzenia := bAdres;
	arModbusOdczytCykliczny[intPetlaPierwszySkan].bFunkcja := TO_BYTE(enumModbusKodyFunkcji.OdczytNRejestrow);
	arModbusOdczytCykliczny[intPetlaPierwszySkan].uiAdresRejestru := 92;
	arModbusOdczytCykliczny[intPetlaPierwszySkan].ltCzestotliwosc := TIME_TO_LTIME(tMinimalnyCzasRaportowania);
	arModbusOdczytCykliczny[intPetlaPierwszySkan].pZmiennaReferencyjna := ADR(wEnergiaCieplnaJednostka);
	intPetlaPierwszySkan := intPetlaPierwszySkan + 1;
	
	arModbusOdczytCykliczny[intPetlaPierwszySkan].bAdresUrzadzenia := bAdres;
	arModbusOdczytCykliczny[intPetlaPierwszySkan].bFunkcja := TO_BYTE(enumModbusKodyFunkcji.OdczytNRejestrow);
	arModbusOdczytCykliczny[intPetlaPierwszySkan].uiAdresRejestru := 82;
	arModbusOdczytCykliczny[intPetlaPierwszySkan].ltCzestotliwosc := TIME_TO_LTIME(tMinimalnyCzasRaportowania);
	arModbusOdczytCykliczny[intPetlaPierwszySkan].pZmiennaReferencyjna := ADR(wPrzeplywJednostka);
	intPetlaPierwszySkan := intPetlaPierwszySkan + 1;
	
	arModbusOdczytCykliczny[intPetlaPierwszySkan].bAdresUrzadzenia := bAdres;
	arModbusOdczytCykliczny[intPetlaPierwszySkan].bFunkcja := TO_BYTE(enumModbusKodyFunkcji.OdczytNRejestrow);
	arModbusOdczytCykliczny[intPetlaPierwszySkan].uiAdresRejestru := 108;
	arModbusOdczytCykliczny[intPetlaPierwszySkan].ltCzestotliwosc := TIME_TO_LTIME(tMinimalnyCzasRaportowania);
	arModbusOdczytCykliczny[intPetlaPierwszySkan].pZmiennaReferencyjna := ADR(wObjetoscJednostka);
	intPetlaPierwszySkan := intPetlaPierwszySkan + 1;
	
	arModbusOdczytCykliczny[intPetlaPierwszySkan].bAdresUrzadzenia := bAdres;
	arModbusOdczytCykliczny[intPetlaPierwszySkan].bFunkcja := TO_BYTE(enumModbusKodyFunkcji.OdczytNRejestrow);
	arModbusOdczytCykliczny[intPetlaPierwszySkan].uiAdresRejestru := 84;
	arModbusOdczytCykliczny[intPetlaPierwszySkan].ltCzestotliwosc := TIME_TO_LTIME(tMinimalnyCzasRaportowania);
	arModbusOdczytCykliczny[intPetlaPierwszySkan].pZmiennaReferencyjna := ADR(wMocJednostka);
	intPetlaPierwszySkan := intPetlaPierwszySkan + 1;
END_IF

// konwersja 2 odczytanych wordów na 32Float
fnKonwersja2x16naFloat32BySchneider(wRejestrMSW := wEnergiaCieplna_Hi, wRejestrLSW := wEnergiaCieplna_Lo, rWartoscFloat32 := rEnergiaCieplna);
fnKonwersja2x16naFloat32BySchneider(wRejestrMSW := wPrzeplyw_Hi, wRejestrLSW := wPrzeplyw_Lo, rWartoscFloat32 := rPrzeplyw);
fnKonwersja2x16naFloat32BySchneider(wRejestrMSW := wObjetosc_Hi, wRejestrLSW := wObjetosc_Lo, rWartoscFloat32 := rObjetosc);
fnKonwersja2x16naFloat32BySchneider(wRejestrMSW := wMoc_Hi, wRejestrLSW := wMoc_Lo, rWartoscFloat32 := rMoc);
fnKonwersja2x16naFloat32BySchneider(wRejestrMSW := wTemperaturaZasilania_Hi, wRejestrLSW := wTemperaturaZasilania_Lo, rWartoscFloat32 := rTemperaturaZasilania);
fnKonwersja2x16naFloat32BySchneider(wRejestrMSW := wTemperaturaPowrotu_Hi, wRejestrLSW := wTemperaturaPowrotu_Lo, rWartoscFloat32 := rTemperaturaPowrotu);

// Przeliczenie zmiennych
fbEnergiaCieplna(	rWartoscWejsciowa := rEnergiaCieplna,
					rDeadband := 100,
					tCzasMinimalny := tMinimalnyCzasRaportowania,
					tCzasMaksymalny := tMaksymalnyCzasRaportowania,
					rWynikMnoznik := 1000000000,
					rWynikOffset := 0,
					rWartoscWejsciowaZaraportowana := rEnergiaCieplnaZaraportowana,
					rWartoscWyjsciowa => rEnergiaCieplna);
					
fbPrzeplyw(	rWartoscWejsciowa := rPrzeplyw,
			rDeadband := 0.00000027778,
			tCzasMinimalny := tMinimalnyCzasRaportowania,
			tCzasMaksymalny := tMaksymalnyCzasRaportowania,
			rWynikMnoznik := 0.00000027778,
			rWynikOffset := 0,
			rWartoscWejsciowaZaraportowana := rPrzeplywZaraportowana,
			rWartoscWyjsciowa => rPrzeplyw);
							
fbObjetosc(	rWartoscWejsciowa := rObjetosc,
			rDeadband := 0.001,
			tCzasMinimalny := tMinimalnyCzasRaportowania,
			tCzasMaksymalny := tMaksymalnyCzasRaportowania,
			rWynikMnoznik := 1,
			rWynikOffset := 0,
			rWartoscWejsciowaZaraportowana := rObjetoscZaraportowana,
			rWartoscWyjsciowa => rObjetosc);								
								
fbMoc(	rWartoscWejsciowa := rMoc,
		rDeadband := 10,
		tCzasMinimalny := tMinimalnyCzasRaportowania,
		tCzasMaksymalny := tMaksymalnyCzasRaportowania,
		rWynikMnoznik := 1000,
		rWynikOffset := 0,
		rWartoscWejsciowaZaraportowana := rMocZaraportowana,
		rWartoscWyjsciowa => rMoc);
				
fbTemperaturaZasilania(	rWartoscWejsciowa := rTemperaturaZasilania,
						rDeadband := 0.1,
						tCzasMinimalny := tMinimalnyCzasRaportowania,
						tCzasMaksymalny := tMaksymalnyCzasRaportowania,
						rWynikMnoznik := 1,
						rWynikOffset := 273.15,
						rWartoscWejsciowaZaraportowana := rTemperaturaZasilaniaZaraportowana,
						rWartoscWyjsciowa => rTemperaturaZasilania);
			
fbTemperaturaPowrotu(	rWartoscWejsciowa := rTemperaturaPowrotu,
						rDeadband := 0.1,
						tCzasMinimalny := tMinimalnyCzasRaportowania,
						tCzasMaksymalny := tMaksymalnyCzasRaportowania,
						rWynikMnoznik := 1,
						rWynikOffset := 273.15,
						rWartoscWejsciowaZaraportowana := rTemperaturaPowrotuZaraportowana,
						rWartoscWyjsciowa => rTemperaturaPowrotu);							

// Sprawdzanie czy pomiar aktualnego przeplywu działa (alarm jest generowany, jeśli odczyt nie zmienił wartości w przeciągu 12h)
IF rPrzeplywPamiec = rPrzeplyw THEN
	xBrakZmianyPrzeplywu := TRUE;
ELSE
	xBrakZmianyPrzeplywu := FALSE;	
END_IF
fbBrakZmianyPrzeplywuTimer(IN := xBrakZmianyPrzeplywu, PT := T#12H);
IF fbBrakZmianyPrzeplywuTimer.Q THEN
	xBladBrakZmianyPrzeplywu := TRUE;
ELSE
	xBladBrakZmianyPrzeplywu := FALSE;
END_IF
rPrzeplywPamiec := rPrzeplyw;

// Sprawdzanie czy pomiar temperatury zasilania działa (alarm jest generowany, jeśli odczyt nie zmienił wartości w przeciągu 12h)
IF rTemperaturaZasilaniaPamiec = rTemperaturaZasilania THEN
	xBrakZmianyTemperaturyZasilania := TRUE;
ELSE
	xBrakZmianyTemperaturyZasilania := FALSE;	
END_IF
fbBrakZmianyTemperaturyZasilaniaTimer(IN := xBrakZmianyTemperaturyZasilania, PT := T#12H);
IF fbBrakZmianyTemperaturyZasilaniaTimer.Q THEN
	xBladBrakZmianyTemperaturyZasilania := TRUE;
ELSE
	xBladBrakZmianyTemperaturyZasilania := FALSE;
END_IF
rTemperaturaZasilaniaPamiec := rTemperaturaZasilania;

// Sprawdzanie czy pomiar temperatury powrotu działa (alarm jest generowany, jeśli odczyt nie zmienił wartości w przeciągu 12h)
IF rTemperaturaPowrotuPamiec = rTemperaturaPowrotu THEN
	xBrakZmianyTemperaturyPowrotu := TRUE;
ELSE
	xBrakZmianyTemperaturyPowrotu := FALSE;	
END_IF
fbBrakZmianyTemperaturyPowrotuTimer(IN := xBrakZmianyTemperaturyPowrotu, PT := T#12H);
IF fbBrakZmianyTemperaturyPowrotuTimer.Q THEN
	xBladBrakZmianyTemperaturyPowrotu := TRUE;
ELSE
	xBladBrakZmianyTemperaturyPowrotu := FALSE;
END_IF
rTemperaturaPowrotuPamiec := rTemperaturaPowrotu;

// Obsluga komunikatu przychodzacego z IZE
IF sKomunikat <> sKomunikatPamiec AND xPoInicjalizacji THEN
	sKomunikatPamiec := sKomunikat;
	IF fnIDOdbiorcyMatch(sKomunikat , sIdInstancji) THEN
		sDane := '';
		//zapytanie typu Q
		IF fnKomunikatTyp(sKomunikat) = 'Q' AND arModbusStatusKomunikacji[bAdres] = enumModbusStatus.KomunikacjaPrawidlowa THEN
			IF fnKomunikatDaneSzukajWartosci(sKomunikat , 'ENCC=') = '?' OR fnKomunikatDaneSzukajWartosci(sKomunikat , 'ALL=') = '?' THEN
				fnKomunikatDaneDodaj_xOverFlow(sDane := sDane , sAtrybut := 'ENCC=' , sWartosc := REAL_TO_STRING(rEnergiaCieplna) , xOverFlow := xOverFlow);	
				IF xOverFlow = TRUE THEN
					fnZapiszKomunikat(	sCalyKomunikat := '' ,
										sTypKomunikatu := 'A' ,
										sMnemonik := sMnemonik ,
										sMACAdres := sMACAdres ,
										sIDNadawcy := sIdInstancji ,
										sIDOdbiorcy := sIdAplikacji ,
										sDaneZapasowe := sDaneZapasowe ,
										sDane := sDane ,
										arTablicaKomunikatow := arTablicaKomunikatow ,
										intTablicaKomunikatowZnacznikZapisu := intTablicaKomunikatowZnacznikZapisu ,
										intTablicaKomunikatowRozmiar := intTablicaKomunikatowRozmiar ,
										sWyslanyKomunikat := sWyslanyKomunikatDummy);
					sDane := '';
				END_IF
			END_IF
			IF fnKomunikatDaneSzukajWartosci(sKomunikat , 'FLOWCC=') = '?' OR fnKomunikatDaneSzukajWartosci(sKomunikat , 'ALL=') = '?' THEN
				fnKomunikatDaneDodaj_xOverFlow(sDane := sDane , sAtrybut := 'FLOWCC=' , sWartosc := REAL_TO_STRING(rPrzeplyw) , xOverFlow := xOverFlow);	
				IF xOverFlow = TRUE THEN
					fnZapiszKomunikat(	sCalyKomunikat := '' ,
										sTypKomunikatu := 'A' ,
										sMnemonik := sMnemonik ,
										sMACAdres := sMACAdres ,
										sIDNadawcy := sIdInstancji ,
										sIDOdbiorcy := sIdAplikacji ,
										sDaneZapasowe := sDaneZapasowe ,
										sDane := sDane ,
										arTablicaKomunikatow := arTablicaKomunikatow ,
										intTablicaKomunikatowZnacznikZapisu := intTablicaKomunikatowZnacznikZapisu ,
										intTablicaKomunikatowRozmiar := intTablicaKomunikatowRozmiar ,
										sWyslanyKomunikat := sWyslanyKomunikatDummy);
					sDane := '';
				END_IF
			END_IF
			IF fnKomunikatDaneSzukajWartosci(sKomunikat , 'VOLCC=') = '?' OR fnKomunikatDaneSzukajWartosci(sKomunikat , 'ALL=') = '?' THEN
				fnKomunikatDaneDodaj_xOverFlow(sDane := sDane , sAtrybut := 'VOLCC=' , sWartosc := REAL_TO_STRING(rObjetosc) , xOverFlow := xOverFlow);	
				IF xOverFlow = TRUE THEN
					fnZapiszKomunikat(	sCalyKomunikat := '' ,
										sTypKomunikatu := 'A' ,
										sMnemonik := sMnemonik ,
										sMACAdres := sMACAdres ,
										sIDNadawcy := sIdInstancji ,
										sIDOdbiorcy := sIdAplikacji ,
										sDaneZapasowe := sDaneZapasowe ,
										sDane := sDane ,
										arTablicaKomunikatow := arTablicaKomunikatow ,
										intTablicaKomunikatowZnacznikZapisu := intTablicaKomunikatowZnacznikZapisu ,
										intTablicaKomunikatowRozmiar := intTablicaKomunikatowRozmiar ,
										sWyslanyKomunikat := sWyslanyKomunikatDummy);
					sDane := '';
				END_IF
			END_IF
			IF fnKomunikatDaneSzukajWartosci(sKomunikat , 'POWCC=') = '?' OR fnKomunikatDaneSzukajWartosci(sKomunikat , 'ALL=') = '?' THEN
				fnKomunikatDaneDodaj_xOverFlow(sDane := sDane , sAtrybut := 'POWCC=' , sWartosc := REAL_TO_STRING(rMoc) , xOverFlow := xOverFlow);	
				IF xOverFlow = TRUE THEN
					fnZapiszKomunikat(	sCalyKomunikat := '' ,
										sTypKomunikatu := 'A' ,
										sMnemonik := sMnemonik ,
										sMACAdres := sMACAdres ,
										sIDNadawcy := sIdInstancji ,
										sIDOdbiorcy := sIdAplikacji ,
										sDaneZapasowe := sDaneZapasowe ,
										sDane := sDane ,
										arTablicaKomunikatow := arTablicaKomunikatow ,
										intTablicaKomunikatowZnacznikZapisu := intTablicaKomunikatowZnacznikZapisu ,
										intTablicaKomunikatowRozmiar := intTablicaKomunikatowRozmiar ,
										sWyslanyKomunikat := sWyslanyKomunikatDummy);
					sDane := '';
				END_IF
			END_IF
			IF fnKomunikatDaneSzukajWartosci(sKomunikat , 'TEMPINCC=') = '?' OR fnKomunikatDaneSzukajWartosci(sKomunikat , 'ALL=') = '?' THEN
				fnKomunikatDaneDodaj_xOverFlow(sDane := sDane , sAtrybut := 'TEMPINCC=' , sWartosc := REAL_TO_STRING(rTemperaturaZasilania) , xOverFlow := xOverFlow);	
				IF xOverFlow = TRUE THEN
					fnZapiszKomunikat(	sCalyKomunikat := '' ,
										sTypKomunikatu := 'A' ,
										sMnemonik := sMnemonik ,
										sMACAdres := sMACAdres ,
										sIDNadawcy := sIdInstancji ,
										sIDOdbiorcy := sIdAplikacji ,
										sDaneZapasowe := sDaneZapasowe ,
										sDane := sDane ,
										arTablicaKomunikatow := arTablicaKomunikatow ,
										intTablicaKomunikatowZnacznikZapisu := intTablicaKomunikatowZnacznikZapisu ,
										intTablicaKomunikatowRozmiar := intTablicaKomunikatowRozmiar ,
										sWyslanyKomunikat := sWyslanyKomunikatDummy);
					sDane := '';
				END_IF
			END_IF
			IF fnKomunikatDaneSzukajWartosci(sKomunikat , 'TEMPOUTCC=') = '?' OR fnKomunikatDaneSzukajWartosci(sKomunikat , 'ALL=') = '?' THEN
				fnKomunikatDaneDodaj_xOverFlow(sDane := sDane , sAtrybut := 'TEMPOUTCC=' , sWartosc := REAL_TO_STRING(rTemperaturaPowrotu) , xOverFlow := xOverFlow);	
				IF xOverFlow = TRUE THEN
					fnZapiszKomunikat(	sCalyKomunikat := '' ,
										sTypKomunikatu := 'A' ,
										sMnemonik := sMnemonik ,
										sMACAdres := sMACAdres ,
										sIDNadawcy := sIdInstancji ,
										sIDOdbiorcy := sIdAplikacji ,
										sDaneZapasowe := sDaneZapasowe ,
										sDane := sDane ,
										arTablicaKomunikatow := arTablicaKomunikatow ,
										intTablicaKomunikatowZnacznikZapisu := intTablicaKomunikatowZnacznikZapisu ,
										intTablicaKomunikatowRozmiar := intTablicaKomunikatowRozmiar ,
										sWyslanyKomunikat := sWyslanyKomunikatDummy);
					sDane := '';
				END_IF
			END_IF
			// Pytanie o stany alarmów
			IF fnKomunikatDaneSzukajWartosci(sKomunikat , 'ALARM=') = '?' OR fnKomunikatDaneSzukajWartosci(sKomunikat , 'ALL=') = '?' THEN
				FOR intPetla := 1 TO 10 BY 1 DO
					// Raportowanie typu E (stanów alarmów) na zapytanie typu Q
					IF arErrorStan[intPetla] <> enumAlarmWartosc.StanNieznany THEN
						fnZapiszKomunikat(	sCalyKomunikat := '' ,
											sTypKomunikatu := 'E' ,
											sMnemonik := sMnemonik ,
											sMACAdres := sMACAdres ,
											sIDNadawcy := sIdInstancji ,
											sIDOdbiorcy := sIdAplikacji ,
											sDaneZapasowe := sDaneZapasowe ,
											sDane := fnKomunikatDaneErrorRetry(xAktywny := arErrorStan[intPetla] = enumAlarmWartosc.StanAlarmowy , intKlasa := arErrorKlasa[intPetla] , intNumer := intPetla),
											arTablicaKomunikatow := arTablicaKomunikatow ,
											intTablicaKomunikatowZnacznikZapisu := intTablicaKomunikatowZnacznikZapisu ,
											intTablicaKomunikatowRozmiar := intTablicaKomunikatowRozmiar ,
											sWyslanyKomunikat := sWyslanyKomunikatDummy);
					END_IF
				END_FOR
			END_IF
		END_IF
		// Raportowanie typu A na zapytanie Q
		IF sDane <> '' THEN
			fnZapiszKomunikat(	sCalyKomunikat := '' ,
								sTypKomunikatu := 'A' ,
								sMnemonik := sMnemonik ,
								sMACAdres := sMACAdres ,
								sIDNadawcy := sIdInstancji ,
								sIDOdbiorcy := sIdAplikacji ,
								sDaneZapasowe := sDaneZapasowe ,
								sDane := sDane ,
								arTablicaKomunikatow := arTablicaKomunikatow ,
								intTablicaKomunikatowZnacznikZapisu := intTablicaKomunikatowZnacznikZapisu ,
								intTablicaKomunikatowRozmiar := intTablicaKomunikatowRozmiar ,
								sWyslanyKomunikat := sWyslanyKomunikatDummy);
		END_IF
	END_IF
END_IF

// Raportowanie typu M do IZE wartosci odczytanych z Modbusa	
IF 	(rPrzeplyw <> rPrzeplywZaraportowana OR rMoc <> rMocZaraportowana OR rEnergiaCieplna <> rEnergiaCieplnaZaraportowana OR rObjetosc <> rObjetoscZaraportowana OR 
	rTemperaturaZasilania <> rTemperaturaZasilaniaZaraportowana OR rTemperaturaPowrotu <> rTemperaturaPowrotuZaraportowana) AND 
	arModbusStatusKomunikacji[bAdres] = enumModbusStatus.KomunikacjaPrawidlowa AND xPoInicjalizacji THEN
	xRaport := TRUE;
END_IF

IF xRaport THEN
	sDane := '';
	xRaport := FALSE;
	// Sumaryczna zużyta energia cieplna licznika
	IF rEnergiaCieplna <> rEnergiaCieplnaZaraportowana THEN
		rEnergiaCieplnaZaraportowana := rEnergiaCieplna;
		fnKomunikatDaneDodaj_xOverFlow(sDane := sDane , sAtrybut := 'ENCC=' , sWartosc := REAL_TO_STRING(rEnergiaCieplna) , xOverFlow := xOverFlow);	
		IF xOverFlow = TRUE THEN
			fnZapiszKomunikat(	sCalyKomunikat := '' ,
								sTypKomunikatu := 'M' ,
								sMnemonik := sMnemonik ,
								sMACAdres := sMACAdres ,
								sIDNadawcy := sIdInstancji ,
								sIDOdbiorcy := sIdAplikacji ,
								sDaneZapasowe := sDaneZapasowe ,
								sDane := sDane ,
								arTablicaKomunikatow := arTablicaKomunikatow ,
								intTablicaKomunikatowZnacznikZapisu := intTablicaKomunikatowZnacznikZapisu ,
								intTablicaKomunikatowRozmiar := intTablicaKomunikatowRozmiar ,
								sWyslanyKomunikat := sWyslanyKomunikatDummy);
			sDane := '';
		END_IF	
	END_IF
	// Biezacy przeplyw licznika 
	IF rPrzeplyw <> rPrzeplywZaraportowana THEN
		rPrzeplywZaraportowana := rPrzeplyw;
		fnKomunikatDaneDodaj_xOverFlow(sDane := sDane , sAtrybut := 'FLOWCC=' , sWartosc := REAL_TO_STRING(rPrzeplyw) , xOverFlow := xOverFlow);	
		IF xOverFlow = TRUE THEN
			fnZapiszKomunikat(	sCalyKomunikat := '' ,
								sTypKomunikatu := 'M' ,
								sMnemonik := sMnemonik ,
								sMACAdres := sMACAdres ,
								sIDNadawcy := sIdInstancji ,
								sIDOdbiorcy := sIdAplikacji ,
								sDaneZapasowe := sDaneZapasowe ,
								sDane := sDane ,
								arTablicaKomunikatow := arTablicaKomunikatow ,
								intTablicaKomunikatowZnacznikZapisu := intTablicaKomunikatowZnacznikZapisu ,
								intTablicaKomunikatowRozmiar := intTablicaKomunikatowRozmiar ,
								sWyslanyKomunikat := sWyslanyKomunikatDummy);
			sDane := '';
		END_IF	
	END_IF
	// Objętość medium, które przepłynęło przez licznik
	IF rObjetosc <> rObjetoscZaraportowana THEN
		rObjetoscZaraportowana := rObjetosc;
		fnKomunikatDaneDodaj_xOverFlow(sDane := sDane , sAtrybut := 'VOLCC=' , sWartosc := REAL_TO_STRING(rObjetosc) , xOverFlow := xOverFlow);	
		IF xOverFlow = TRUE THEN
			fnZapiszKomunikat(	sCalyKomunikat := '' ,
								sTypKomunikatu := 'M' ,
								sMnemonik := sMnemonik ,
								sMACAdres := sMACAdres ,
								sIDNadawcy := sIdInstancji ,
								sIDOdbiorcy := sIdAplikacji ,
								sDaneZapasowe := sDaneZapasowe ,
								sDane := sDane ,
								arTablicaKomunikatow := arTablicaKomunikatow ,
								intTablicaKomunikatowZnacznikZapisu := intTablicaKomunikatowZnacznikZapisu ,
								intTablicaKomunikatowRozmiar := intTablicaKomunikatowRozmiar ,
								sWyslanyKomunikat := sWyslanyKomunikatDummy);
			sDane := '';
		END_IF	
	END_IF
	// Biezaca moc licznika
	IF rMoc <> rMocZaraportowana THEN
		rMocZaraportowana := rMoc;
		fnKomunikatDaneDodaj_xOverFlow(sDane := sDane , sAtrybut := 'POWCC=' , sWartosc := REAL_TO_STRING(rMoc) , xOverFlow := xOverFlow);	
		IF xOverFlow = TRUE THEN
			fnZapiszKomunikat(	sCalyKomunikat := '' ,
								sTypKomunikatu := 'M' ,
								sMnemonik := sMnemonik ,
								sMACAdres := sMACAdres ,
								sIDNadawcy := sIdInstancji ,
								sIDOdbiorcy := sIdAplikacji ,
								sDaneZapasowe := sDaneZapasowe ,
								sDane := sDane ,
								arTablicaKomunikatow := arTablicaKomunikatow ,
								intTablicaKomunikatowZnacznikZapisu := intTablicaKomunikatowZnacznikZapisu ,
								intTablicaKomunikatowRozmiar := intTablicaKomunikatowRozmiar ,
								sWyslanyKomunikat := sWyslanyKomunikatDummy);
			sDane := '';
		END_IF	
	END_IF
	// Temperatura na wejsciu licznika
	IF rTemperaturaZasilania <> rTemperaturaZasilaniaZaraportowana THEN
		rTemperaturaZasilaniaZaraportowana := rTemperaturaZasilania;
		fnKomunikatDaneDodaj_xOverFlow(sDane := sDane , sAtrybut := 'TEMPINCC=' , sWartosc := REAL_TO_STRING(rTemperaturaZasilania) , xOverFlow := xOverFlow);	
		IF xOverFlow = TRUE THEN
			fnZapiszKomunikat(	sCalyKomunikat := '' ,
								sTypKomunikatu := 'M' ,
								sMnemonik := sMnemonik ,
								sMACAdres := sMACAdres ,
								sIDNadawcy := sIdInstancji ,
								sIDOdbiorcy := sIdAplikacji ,
								sDaneZapasowe := sDaneZapasowe ,
								sDane := sDane ,
								arTablicaKomunikatow := arTablicaKomunikatow ,
								intTablicaKomunikatowZnacznikZapisu := intTablicaKomunikatowZnacznikZapisu ,
								intTablicaKomunikatowRozmiar := intTablicaKomunikatowRozmiar ,
								sWyslanyKomunikat := sWyslanyKomunikatDummy);
			sDane := '';
		END_IF	
	END_IF
		// Temperatura na wyjsciu licznika
	IF rTemperaturaPowrotu <> rTemperaturaPowrotuZaraportowana THEN
		rTemperaturaPowrotuZaraportowana := rTemperaturaPowrotu;
		fnKomunikatDaneDodaj_xOverFlow(sDane := sDane , sAtrybut := 'TEMPOUTCC=' , sWartosc := REAL_TO_STRING(rTemperaturaPowrotu) , xOverFlow := xOverFlow);	
		IF xOverFlow = TRUE THEN
			fnZapiszKomunikat(	sCalyKomunikat := '' ,
								sTypKomunikatu := 'M' ,
								sMnemonik := sMnemonik ,
								sMACAdres := sMACAdres ,
								sIDNadawcy := sIdInstancji ,
								sIDOdbiorcy := sIdAplikacji ,
								sDaneZapasowe := sDaneZapasowe ,
								sDane := sDane ,
								arTablicaKomunikatow := arTablicaKomunikatow ,
								intTablicaKomunikatowZnacznikZapisu := intTablicaKomunikatowZnacznikZapisu ,
								intTablicaKomunikatowRozmiar := intTablicaKomunikatowRozmiar ,
								sWyslanyKomunikat := sWyslanyKomunikatDummy);
			sDane := '';
		END_IF	
	END_IF
	
	IF sDane <> '' AND xPoInicjalizacji THEN
		fnZapiszKomunikat(	sCalyKomunikat := '' ,
							sTypKomunikatu := 'M' ,
							sMnemonik := sMnemonik ,
							sMACAdres := sMACAdres ,
							sIDNadawcy := sIdInstancji ,
							sIDOdbiorcy := sIdAplikacji ,
							sDaneZapasowe := sDaneZapasowe ,
							sDane := sDane ,
							arTablicaKomunikatow := arTablicaKomunikatow ,
							intTablicaKomunikatowZnacznikZapisu := intTablicaKomunikatowZnacznikZapisu ,
							intTablicaKomunikatowRozmiar := intTablicaKomunikatowRozmiar ,
							sWyslanyKomunikat := sWyslanyKomunikat);
	END_IF
END_IF
	
// Alarm braku komunikacji MODBUS 
IF arErrorStan[enumPPPSLicznikCieplaMultical403Error.BrakKomunikacji] <> enumAlarmWartosc.StanAlarmowy AND arModbusStatusKomunikacji[bAdres] = enumModbusStatus.BrakKomunikacji THEN
	arErrorStan[enumPPPSLicznikCieplaMultical403Error.BrakKomunikacji] := enumAlarmWartosc.StanAlarmowy;
	arErrorKlasa[enumPPPSLicznikCieplaMultical403Error.BrakKomunikacji] := enumPPPSLicznikCieplaMultical403Error.BrakKomunikacji;
	IF xPoInicjalizacji THEN
		fnZapiszKomunikat(	sCalyKomunikat := '',
							sTypKomunikatu := 'E',
							sMnemonik := sMnemonik,
							sMACAdres := sMACAdres,
							sIDNadawcy := sIdInstancji,
							sIDOdbiorcy := sIdAplikacji,
							sDaneZapasowe := sDaneZapasowe,
							sDane := fnKomunikatDaneError(	xAktywny := TRUE, 
															intKlasa := enumPPPSLicznikCieplaMultical403ErrorKlasa.BrakKomunikacji, 
															intNumer := enumPPPSLicznikCieplaMultical403Error.BrakKomunikacji),
							arTablicaKomunikatow := arTablicaKomunikatow,
							intTablicaKomunikatowZnacznikZapisu := intTablicaKomunikatowZnacznikZapisu,
							intTablicaKomunikatowRozmiar := intTablicaKomunikatowRozmiar,
							sWyslanyKomunikat := sWyslanyKomunikatDummy);
	END_IF
END_IF
IF arErrorStan[enumPPPSLicznikCieplaMultical403Error.BrakKomunikacji] <> enumAlarmWartosc.StanNormalny AND arModbusStatusKomunikacji[bAdres] = enumModbusStatus.KomunikacjaPrawidlowa THEN
	arErrorStan[enumPPPSLicznikCieplaMultical403Error.BrakKomunikacji] := enumAlarmWartosc.StanNormalny;
	arErrorKlasa[enumPPPSLicznikCieplaMultical403Error.BrakKomunikacji] := enumPPPSLicznikCieplaMultical403Error.BrakKomunikacji;
	IF xPoInicjalizacji THEN
		fnZapiszKomunikat(	sCalyKomunikat := '',
							sTypKomunikatu := 'E',
							sMnemonik := sMnemonik,
							sMACAdres := sMACAdres,
							sIDNadawcy := sIdInstancji,
							sIDOdbiorcy := sIdAplikacji,
							sDaneZapasowe := sDaneZapasowe,
							sDane := fnKomunikatDaneError(	xAktywny := FALSE, 
															intKlasa := enumPPPSLicznikCieplaMultical403ErrorKlasa.BrakKomunikacji, 
															intNumer := enumPPPSLicznikCieplaMultical403Error.BrakKomunikacji),
							arTablicaKomunikatow := arTablicaKomunikatow,
							intTablicaKomunikatowZnacznikZapisu := intTablicaKomunikatowZnacznikZapisu,
							intTablicaKomunikatowRozmiar := intTablicaKomunikatowRozmiar,
							sWyslanyKomunikat := sWyslanyKomunikatDummy);
	END_IF
END_IF
	
// Alarm czujnika przepływu
IF arErrorStan[enumPPPSLicznikCieplaMultical403Error.AlarmCzujnikaPrzeplywu] <> enumAlarmWartosc.StanAlarmowy AND xBladBrakZmianyPrzeplywu THEN
	arErrorStan[enumPPPSLicznikCieplaMultical403Error.AlarmCzujnikaPrzeplywu] := enumAlarmWartosc.StanAlarmowy;
	arErrorKlasa[enumPPPSLicznikCieplaMultical403Error.AlarmCzujnikaPrzeplywu] := enumPPPSLicznikCieplaMultical403Error.AlarmCzujnikaPrzeplywu;
	IF xPoInicjalizacji THEN
		fnZapiszKomunikat(	sCalyKomunikat := '',
							sTypKomunikatu := 'E',
							sMnemonik := sMnemonik,
							sMACAdres := sMACAdres,
							sIDNadawcy := sIdInstancji,
							sIDOdbiorcy := sIdAplikacji,
							sDaneZapasowe := sDaneZapasowe,
							sDane := fnKomunikatDaneError(	xAktywny := TRUE, 
															intKlasa := enumPPPSLicznikCieplaMultical403ErrorKlasa.AlarmCzujnikaPrzeplywu, 
															intNumer := enumPPPSLicznikCieplaMultical403Error.AlarmCzujnikaPrzeplywu),
							arTablicaKomunikatow := arTablicaKomunikatow,
							intTablicaKomunikatowZnacznikZapisu := intTablicaKomunikatowZnacznikZapisu,
							intTablicaKomunikatowRozmiar := intTablicaKomunikatowRozmiar,
							sWyslanyKomunikat := sWyslanyKomunikatDummy);
	END_IF
END_IF
IF arErrorStan[enumPPPSLicznikCieplaMultical403Error.AlarmCzujnikaPrzeplywu] <> enumAlarmWartosc.StanNormalny AND NOT xBladBrakZmianyPrzeplywu THEN
	arErrorStan[enumPPPSLicznikCieplaMultical403Error.AlarmCzujnikaPrzeplywu] := enumAlarmWartosc.StanNormalny;
	arErrorKlasa[enumPPPSLicznikCieplaMultical403Error.AlarmCzujnikaPrzeplywu] := enumPPPSLicznikCieplaMultical403Error.AlarmCzujnikaPrzeplywu;
	IF xPoInicjalizacji THEN
		fnZapiszKomunikat(	sCalyKomunikat := '',
							sTypKomunikatu := 'E',
							sMnemonik := sMnemonik,
							sMACAdres := sMACAdres,
							sIDNadawcy := sIdInstancji,
							sIDOdbiorcy := sIdAplikacji,
							sDaneZapasowe := sDaneZapasowe,
							sDane := fnKomunikatDaneError(	xAktywny := FALSE, 
															intKlasa := enumPPPSLicznikCieplaMultical403ErrorKlasa.AlarmCzujnikaPrzeplywu, 
															intNumer := enumPPPSLicznikCieplaMultical403Error.AlarmCzujnikaPrzeplywu),
							arTablicaKomunikatow := arTablicaKomunikatow,
							intTablicaKomunikatowZnacznikZapisu := intTablicaKomunikatowZnacznikZapisu,
							intTablicaKomunikatowRozmiar := intTablicaKomunikatowRozmiar ,
							sWyslanyKomunikat := sWyslanyKomunikatDummy);
	END_IF
END_IF
	
// Alarm czujnika temperatury zasilania
IF arErrorStan[enumPPPSLicznikCieplaMultical403Error.AlarmCzujnikaZasilania] <> enumAlarmWartosc.StanAlarmowy AND xBladBrakZmianyTemperaturyZasilania THEN
	arErrorStan[enumPPPSLicznikCieplaMultical403Error.AlarmCzujnikaZasilania] := enumAlarmWartosc.StanAlarmowy;
	arErrorKlasa[enumPPPSLicznikCieplaMultical403Error.AlarmCzujnikaZasilania] := enumPPPSLicznikCieplaMultical403Error.AlarmCzujnikaZasilania;
	IF xPoInicjalizacji THEN
		fnZapiszKomunikat(	sCalyKomunikat := '',
							sTypKomunikatu := 'E',
							sMnemonik := sMnemonik,
							sMACAdres := sMACAdres,
							sIDNadawcy := sIdInstancji,
							sIDOdbiorcy := sIdAplikacji,
							sDaneZapasowe := sDaneZapasowe,
							sDane := fnKomunikatDaneError(	xAktywny := TRUE, 
														  	intKlasa := enumPPPSLicznikCieplaMultical403ErrorKlasa.AlarmCzujnikaZasilania, 
															intNumer := enumPPPSLicznikCieplaMultical403Error.AlarmCzujnikaZasilania),
							arTablicaKomunikatow := arTablicaKomunikatow,
							intTablicaKomunikatowZnacznikZapisu := intTablicaKomunikatowZnacznikZapisu,
							intTablicaKomunikatowRozmiar := intTablicaKomunikatowRozmiar,
							sWyslanyKomunikat := sWyslanyKomunikatDummy);
	END_IF
END_IF
IF arErrorStan[enumPPPSLicznikCieplaMultical403Error.AlarmCzujnikaZasilania] <> enumAlarmWartosc.StanNormalny AND NOT xBladBrakZmianyTemperaturyZasilania THEN
	arErrorStan[enumPPPSLicznikCieplaMultical403Error.AlarmCzujnikaZasilania] := enumAlarmWartosc.StanNormalny;
	arErrorKlasa[enumPPPSLicznikCieplaMultical403Error.AlarmCzujnikaZasilania] := enumPPPSLicznikCieplaMultical403Error.AlarmCzujnikaZasilania;
	IF xPoInicjalizacji THEN
		fnZapiszKomunikat(	sCalyKomunikat := '',
							sTypKomunikatu := 'E',
							sMnemonik := sMnemonik,
							sMACAdres := sMACAdres,
							sIDNadawcy := sIdInstancji,
							sIDOdbiorcy := sIdAplikacji,
							sDaneZapasowe := sDaneZapasowe,
							sDane := fnKomunikatDaneError(	xAktywny := FALSE, 
															intKlasa := enumPPPSLicznikCieplaMultical403ErrorKlasa.AlarmCzujnikaZasilania, 
															intNumer := enumPPPSLicznikCieplaMultical403Error.AlarmCzujnikaZasilania),
							arTablicaKomunikatow := arTablicaKomunikatow,
							intTablicaKomunikatowZnacznikZapisu := intTablicaKomunikatowZnacznikZapisu,
							intTablicaKomunikatowRozmiar := intTablicaKomunikatowRozmiar ,
							sWyslanyKomunikat := sWyslanyKomunikatDummy);
	END_IF
END_IF	
	
// Alarm czujnika temperatury powrotu
IF arErrorStan[enumPPPSLicznikCieplaMultical403Error.AlarmCzujnikaPowrotu] <> enumAlarmWartosc.StanAlarmowy AND xBladBrakZmianyTemperaturyPowrotu THEN
	arErrorStan[enumPPPSLicznikCieplaMultical403Error.AlarmCzujnikaPowrotu] := enumAlarmWartosc.StanAlarmowy;
	arErrorKlasa[enumPPPSLicznikCieplaMultical403Error.AlarmCzujnikaPowrotu] := enumPPPSLicznikCieplaMultical403Error.AlarmCzujnikaPowrotu;
	IF xPoInicjalizacji THEN
		fnZapiszKomunikat(	sCalyKomunikat := '',
							sTypKomunikatu := 'E',
							sMnemonik := sMnemonik,
							sMACAdres := sMACAdres,
							sIDNadawcy := sIdInstancji,
							sIDOdbiorcy := sIdAplikacji,
							sDaneZapasowe := sDaneZapasowe,
							sDane := fnKomunikatDaneError(	xAktywny := TRUE, 
															intKlasa := enumPPPSLicznikCieplaMultical403ErrorKlasa.AlarmCzujnikaPowrotu, 
															intNumer := enumPPPSLicznikCieplaMultical403Error.AlarmCzujnikaPowrotu),
							arTablicaKomunikatow := arTablicaKomunikatow,
							intTablicaKomunikatowZnacznikZapisu := intTablicaKomunikatowZnacznikZapisu,
							intTablicaKomunikatowRozmiar := intTablicaKomunikatowRozmiar,
							sWyslanyKomunikat := sWyslanyKomunikatDummy);
	END_IF
END_IF
IF arErrorStan[enumPPPSLicznikCieplaMultical403Error.AlarmCzujnikaPowrotu] <> enumAlarmWartosc.StanNormalny AND NOT xBladBrakZmianyTemperaturyPowrotu THEN
	arErrorStan[enumPPPSLicznikCieplaMultical403Error.AlarmCzujnikaPowrotu] := enumAlarmWartosc.StanNormalny;
	arErrorKlasa[enumPPPSLicznikCieplaMultical403Error.AlarmCzujnikaPowrotu] := enumPPPSLicznikCieplaMultical403Error.AlarmCzujnikaPowrotu;
	IF xPoInicjalizacji THEN
		fnZapiszKomunikat(	sCalyKomunikat := '',
							sTypKomunikatu := 'E',
							sMnemonik := sMnemonik,
							sMACAdres := sMACAdres,
							sIDNadawcy := sIdInstancji,
							sIDOdbiorcy := sIdAplikacji,
							sDaneZapasowe := sDaneZapasowe,
							sDane := fnKomunikatDaneError(	xAktywny := FALSE, 
															intKlasa := enumPPPSLicznikCieplaMultical403ErrorKlasa.AlarmCzujnikaPowrotu, 
															intNumer := enumPPPSLicznikCieplaMultical403Error.AlarmCzujnikaPowrotu),
							arTablicaKomunikatow := arTablicaKomunikatow,
							intTablicaKomunikatowZnacznikZapisu := intTablicaKomunikatowZnacznikZapisu,
							intTablicaKomunikatowRozmiar := intTablicaKomunikatowRozmiar ,
							sWyslanyKomunikat := sWyslanyKomunikatDummy);
	END_IF
END_IF
	
          
END_FUNCTION_BLOCK

FUNCTION_BLOCK fbPPPSLicznikCieplaMultical602
  VAR_INPUT
    sKomunikat : alSTRINGKomunikat;  (* komunikat z systemu zewnętrznego *)
    intTablicaKomunikatowRozmiar : INT;  (* rozmiar tablicy danych wysyłkowych *)
    intModbusOdczytZapisZadanieRozmiar : INT;  (* rozmiar tablicy danych modbusa *)
    xTablicaKomunikatowHold : BOOL;  (* wstrzymanie komunikacji mniej ważnych komunikatów *)
    sIdInstancji : STRING;  (* parametr ID rolety np NS02L*202IBM**** *)
    sIdAplikacji : STRING;  (* parametr ID aplikacji np SO*******ECL*000 *)
    sMnemonik : STRING;  (* mnemonik właściciela - BCB* *)
    sMACAdres : STRING;  (* MAC adres sterownika *)
    sDaneZapasowe : STRING;  (* 6 znaków zapasu *)
    tCzasOpoznieniaRestartu : TIME;  (* czas opóźnienia po którym zaczynają być raportowane wartości *)
    tCzasOpoznieniaAlarmu : TIME := TIME#1m0s0ms;  (* czas opóźnienia po którym zaczynają być raportowane wartości *)
    bAdres : BYTE;
    tMinimalnyCzasRaportowania : TIME;
    tMaksymalnyCzasRaportowania : TIME;
    xAutonomizacja : BOOL;
    xAutonomizacjaSztuczna : BOOL;
  END_VAR
  VAR_IN_OUT
    arModbusOdczytCykliczny : ARRAY[1..5000] OF typModbusOdczytCykliczny;
    arModbusStatusKomunikacji : ARRAY[1..256] OF INT;
    arTablicaKomunikatow : alARRAYTablicaKomunikatow;
    intTablicaKomunikatowZnacznikZapisu : INT;
  END_VAR
  VAR
    xPoInicjalizacji : BOOL := FALSE;  (* Inicjalizacja *)
    fbInicjalizacyjnyTimer : TON;
    tCzasInicjalizacji : TIME := TIME#30s0ms;
    xPierwszySkan : BOOL := TRUE;  (* Definicje zmiennych do odczytu wartości z modbusa *)
    intPetlaPierwszySkan : INT := 1;
    sDane : alSTRINGKomunikat;  (* Definicje do komunikacji z IZE *)
    sWyslanyKomunikat : alSTRINGKomunikat;
    sWyslanyKomunikatDummy : alSTRINGKomunikat;
    xZadanieRaportu : BOOL;
    sKomunikatPamiec : alSTRINGKomunikat;
    intPetla : INT;
    arErrorStan : ARRAY[0..10] OF INT;  (* tablica przechowująca statusy alarmowe *)
    arErrorKlasa : ARRAY[0..10] OF INT;  (* tablica przechowująca klasy danych alarmów *)
    xRaport : BOOL := FALSE;
    sTempWartoscAtrybutu : STRING;
    xOverFlow : BOOL;
    fbTimerBrakuKomunikacji : TON;  (* Kontrola komunikacji urządzenia *)
    xBrakKomunikacjiPLC : BOOL;
    xBrakKomunikacjiIZE : BOOL;
    wEnergiaCieplna_Lo : WORD;  (* Całkowita energia cieplna *)
    wEnergiaCieplna_Hi : WORD;
    rEnergiaCieplna : REAL;
    fbEnergiaCieplna : fbFiltrWartoscAnalogowa;
    rEnergiaCieplnaZaraportowana : REAL;
    wEnergiaCieplnaJednostka : WORD;  (* Jednostka energii cieplnej *)
    wPrzeplyw_Lo : WORD;  (* Aktualna wartość przepływu *)
    wPrzeplyw_Hi : WORD;
    rPrzeplyw : REAL;
    fbPrzeplyw : fbFiltrWartoscAnalogowa;
    rPrzeplywZaraportowana : REAL;
    wPrzeplywJednostka : REAL;  (* Jednostka przepływu *)
    rPrzeplywPamiec : REAL;  (* Wartosc przechowywana w pamieci w celu porównania z wartością aktualną *)
    xBrakZmianyPrzeplywu : BOOL;  (* Flaga informująca o braku zmiany przepływu w czasie *)
    fbBrakZmianyPrzeplywuTimer : TON;
    xBladBrakZmianyPrzeplywu : BOOL;  (* Flaga informująca o braku przeplywu przez czas 12h - podstawa wygenerowania alarmu *)
    wObjetosc_Lo : WORD;  (* Objętość medium, które przepłynęło przez licznik *)
    wObjetosc_Hi : WORD;
    rObjetosc : REAL;
    fbObjetosc : fbFiltrWartoscAnalogowa;
    rObjetoscZaraportowana : REAL;
    wObjetoscJednostka : WORD;  (* Jednostka wolumenu *)
    wMoc_Hi : WORD;  (* Aktualna moc cieplna płynąca przez licznik *)
    wMoc_Lo : WORD;
    rMoc : REAL;
    fbMoc : fbFiltrWartoscAnalogowa;
    rMocZaraportowana : REAL;
    wMocJednostka : WORD;  (* Jednostka mocy *)
    wTemperaturaZasilania_Lo : WORD;  (* Temp czynnika na wejściu licznika *)
    wTemperaturaZasilania_Hi : WORD;
    rTemperaturaZasilania : REAL;
    fbTemperaturaZasilania : fbFiltrWartoscAnalogowa;
    rTemperaturaZasilaniaZaraportowana : REAL;
    rTemperaturaZasilaniaPamiec : REAL;  (* Wartosc przechowywana w pamieci w celu porównania z wartością aktualną *)
    xBrakZmianyTemperaturyZasilania : BOOL;  (* Flaga informująca o braku zmiany przepływu w czasie *)
    fbBrakZmianyTemperaturyZasilaniaTimer : TON;
    xBladBrakZmianyTemperaturyZasilania : BOOL;  (* Flaga informująca o braku przeplywu przez czas 12h - podstawa wygenerowania alarmu *)
    wTemperaturaPowrotu_Lo : WORD;  (* Temp czynnika na wyjściu licznika *)
    wTemperaturaPowrotu_Hi : WORD;
    rTemperaturaPowrotu : REAL;
    fbTemperaturaPowrotu : fbFiltrWartoscAnalogowa;
    rTemperaturaPowrotuZaraportowana : REAL;
    rTemperaturaPowrotuPamiec : REAL;  (* Wartosc przechowywana w pamieci w celu porównania z wartością aktualną *)
    xBrakZmianyTemperaturyPowrotu : BOOL;  (* Flaga informująca o braku zmiany przepływu w czasie *)
    fbBrakZmianyTemperaturyPowrotuTimer : TON;
    xBladBrakZmianyTemperaturyPowrotu : BOOL;  (* Flaga informująca o braku przeplywu przez czas 12h - podstawa wygenerowania alarmu *)
  END_VAR

            (*			
Autor:					Jan Cichosz, 2019-03-25 
Prawa majątkowe: 		Solwena Sp. z o.o., 
Aktualizacje:			2019-05-16-AWy: Modyfikacja warunku na raportowanie. Dopisane: AND arModbusStatusKomunikacji[bAdres] = enumModbusStatus.KomunikacjaPrawidlowa AND xPoInicjalizacji
						2019-05-16-JC: Poprawki w formatowaniu, zmiany nazw zmiennych 
						2019-08-08-AWy: Zmiana nazw zmiennych i usunięcie zbędnych. Poprawki przy przeliczaniu zmiennych. Poprwaki w nazwach atrybutów. Generowanie alarmów czujników temperatury.
										Wysyłanie alarmów. Usunięcie blokady wykonywania rozkazów.
						2019-08-29-AWy: Zmiana poszczególnych parametrów przy przeliczaniu zmiennych. Usunięcie buga z raporotwania mocy.
					
Opis:					Komunikacja z licznikami ciepła Multical 602							
*)

// Inicjalizacja sterownika
fbInicjalizacyjnyTimer(IN := (NOT xPoInicjalizacji AND arModbusStatusKomunikacji[bAdres] = enumModbusStatus.KomunikacjaPrawidlowa), PT := tCzasOpoznieniaRestartu);
IF fbInicjalizacyjnyTimer.Q THEN
	rPrzeplywZaraportowana := rPrzeplyw;
	rMocZaraportowana := rMoc;
	rEnergiaCieplnaZaraportowana := rEnergiaCieplna;
	rObjetoscZaraportowana := rObjetosc;
	rTemperaturaZasilaniaZaraportowana := rTemperaturaZasilania;
	rTemperaturaPowrotuZaraportowana := rTemperaturaPowrotu;
	xPoInicjalizacji := TRUE;
END_IF
mirek jest Słaby

// Włącz autonomizację jeśli sterownik jest w stanie inicjalizacji lub nastąpiło wymuszenie autonomizacji
IF NOT xPoInicjalizacji OR xAutonomizacjaSztuczna = TRUE THEN
	xAutonomizacja := TRUE;
END_IF 

// Kontrola komunikacji
fbTimerBrakuKomunikacji(IN := arModbusStatusKomunikacji[bAdres] = enumModbusStatus.BrakKomunikacji, PT := T#60S);
IF fbTimerBrakuKomunikacji.Q THEN
	xBrakKomunikacjiPLC := TRUE;
ELSE
	xBrakKomunikacjiPLC := FALSE;
END_IF

IF xAutonomizacja THEN
	xBrakKomunikacjiIZE := TRUE;
ELSE
	xBrakKomunikacjiIZE := FALSE;
END_IF

// Deklaracja rejestrów Modbusa
IF xPierwszySkan THEN
	xPierwszySkan := FALSE;
	WHILE arModbusOdczytCykliczny[intPetlaPierwszySkan].bAdresUrzadzenia <> 0 DO
		intPetlaPierwszySkan := intPetlaPierwszySkan + 1;
	END_WHILE
	arModbusOdczytCykliczny[intPetlaPierwszySkan].bAdresUrzadzenia := bAdres;
	arModbusOdczytCykliczny[intPetlaPierwszySkan].bFunkcja := TO_BYTE(enumModbusKodyFunkcji.OdczytNRejestrow);
	arModbusOdczytCykliczny[intPetlaPierwszySkan].uiAdresRejestru := 256;
	arModbusOdczytCykliczny[intPetlaPierwszySkan].ltCzestotliwosc := TIME_TO_LTIME(tMinimalnyCzasRaportowania);
	arModbusOdczytCykliczny[intPetlaPierwszySkan].pZmiennaReferencyjna := ADR(wEnergiaCieplna_Hi);
	intPetlaPierwszySkan := intPetlaPierwszySkan + 1;	
	
	arModbusOdczytCykliczny[intPetlaPierwszySkan].bAdresUrzadzenia := bAdres;
	arModbusOdczytCykliczny[intPetlaPierwszySkan].bFunkcja := TO_BYTE(enumModbusKodyFunkcji.OdczytNRejestrow);
	arModbusOdczytCykliczny[intPetlaPierwszySkan].uiAdresRejestru := 257;
	arModbusOdczytCykliczny[intPetlaPierwszySkan].ltCzestotliwosc := TIME_TO_LTIME(tMinimalnyCzasRaportowania);
	arModbusOdczytCykliczny[intPetlaPierwszySkan].pZmiennaReferencyjna := ADR(wEnergiaCieplna_Lo);
	intPetlaPierwszySkan := intPetlaPierwszySkan + 1;
	
	arModbusOdczytCykliczny[intPetlaPierwszySkan].bAdresUrzadzenia := bAdres;
	arModbusOdczytCykliczny[intPetlaPierwszySkan].bFunkcja := TO_BYTE(enumModbusKodyFunkcji.OdczytNRejestrow);
	arModbusOdczytCykliczny[intPetlaPierwszySkan].uiAdresRejestru := 258;
	arModbusOdczytCykliczny[intPetlaPierwszySkan].ltCzestotliwosc := TIME_TO_LTIME(tMinimalnyCzasRaportowania);
	arModbusOdczytCykliczny[intPetlaPierwszySkan].pZmiennaReferencyjna := ADR(wPrzeplyw_Hi);
	intPetlaPierwszySkan := intPetlaPierwszySkan + 1;

	arModbusOdczytCykliczny[intPetlaPierwszySkan].bAdresUrzadzenia := bAdres;
	arModbusOdczytCykliczny[intPetlaPierwszySkan].bFunkcja := TO_BYTE(enumModbusKodyFunkcji.OdczytNRejestrow);
	arModbusOdczytCykliczny[intPetlaPierwszySkan].uiAdresRejestru := 259;
	arModbusOdczytCykliczny[intPetlaPierwszySkan].ltCzestotliwosc := TIME_TO_LTIME(tMinimalnyCzasRaportowania);
	arModbusOdczytCykliczny[intPetlaPierwszySkan].pZmiennaReferencyjna := ADR(wPrzeplyw_Lo);
	intPetlaPierwszySkan := intPetlaPierwszySkan + 1;
	
	arModbusOdczytCykliczny[intPetlaPierwszySkan].bAdresUrzadzenia := bAdres;
	arModbusOdczytCykliczny[intPetlaPierwszySkan].bFunkcja := TO_BYTE(enumModbusKodyFunkcji.OdczytNRejestrow);
	arModbusOdczytCykliczny[intPetlaPierwszySkan].uiAdresRejestru := 260;
	arModbusOdczytCykliczny[intPetlaPierwszySkan].ltCzestotliwosc := TIME_TO_LTIME(tMinimalnyCzasRaportowania);
	arModbusOdczytCykliczny[intPetlaPierwszySkan].pZmiennaReferencyjna := ADR(wObjetosc_Hi);
	intPetlaPierwszySkan := intPetlaPierwszySkan + 1;
	
	arModbusOdczytCykliczny[intPetlaPierwszySkan].bAdresUrzadzenia := bAdres;
	arModbusOdczytCykliczny[intPetlaPierwszySkan].bFunkcja := TO_BYTE(enumModbusKodyFunkcji.OdczytNRejestrow);
	arModbusOdczytCykliczny[intPetlaPierwszySkan].uiAdresRejestru := 261;
	arModbusOdczytCykliczny[intPetlaPierwszySkan].ltCzestotliwosc := TIME_TO_LTIME(tMinimalnyCzasRaportowania);
	arModbusOdczytCykliczny[intPetlaPierwszySkan].pZmiennaReferencyjna := ADR(wObjetosc_Lo);
	intPetlaPierwszySkan := intPetlaPierwszySkan + 1;
	
	arModbusOdczytCykliczny[intPetlaPierwszySkan].bAdresUrzadzenia := bAdres;
	arModbusOdczytCykliczny[intPetlaPierwszySkan].bFunkcja := TO_BYTE(enumModbusKodyFunkcji.OdczytNRejestrow);
	arModbusOdczytCykliczny[intPetlaPierwszySkan].uiAdresRejestru := 262;
	arModbusOdczytCykliczny[intPetlaPierwszySkan].ltCzestotliwosc := TIME_TO_LTIME(tMinimalnyCzasRaportowania);
	arModbusOdczytCykliczny[intPetlaPierwszySkan].pZmiennaReferencyjna := ADR(wMoc_Hi);
	intPetlaPierwszySkan := intPetlaPierwszySkan + 1;	
	
	arModbusOdczytCykliczny[intPetlaPierwszySkan].bAdresUrzadzenia := bAdres;
	arModbusOdczytCykliczny[intPetlaPierwszySkan].bFunkcja := TO_BYTE(enumModbusKodyFunkcji.OdczytNRejestrow);
	arModbusOdczytCykliczny[intPetlaPierwszySkan].uiAdresRejestru := 263;
	arModbusOdczytCykliczny[intPetlaPierwszySkan].ltCzestotliwosc := TIME_TO_LTIME(tMinimalnyCzasRaportowania);
	arModbusOdczytCykliczny[intPetlaPierwszySkan].pZmiennaReferencyjna := ADR(wMoc_Lo);
	intPetlaPierwszySkan := intPetlaPierwszySkan + 1;
	
	arModbusOdczytCykliczny[intPetlaPierwszySkan].bAdresUrzadzenia := bAdres;
	arModbusOdczytCykliczny[intPetlaPierwszySkan].bFunkcja := TO_BYTE(enumModbusKodyFunkcji.OdczytNRejestrow);
	arModbusOdczytCykliczny[intPetlaPierwszySkan].uiAdresRejestru := 264;
	arModbusOdczytCykliczny[intPetlaPierwszySkan].ltCzestotliwosc := TIME_TO_LTIME(tMinimalnyCzasRaportowania);
	arModbusOdczytCykliczny[intPetlaPierwszySkan].pZmiennaReferencyjna := ADR(wTemperaturaZasilania_Hi);
	intPetlaPierwszySkan := intPetlaPierwszySkan + 1;	
	
	arModbusOdczytCykliczny[intPetlaPierwszySkan].bAdresUrzadzenia := bAdres;
	arModbusOdczytCykliczny[intPetlaPierwszySkan].bFunkcja := TO_BYTE(enumModbusKodyFunkcji.OdczytNRejestrow);
	arModbusOdczytCykliczny[intPetlaPierwszySkan].uiAdresRejestru := 265;
	arModbusOdczytCykliczny[intPetlaPierwszySkan].ltCzestotliwosc := TIME_TO_LTIME(tMinimalnyCzasRaportowania);
	arModbusOdczytCykliczny[intPetlaPierwszySkan].pZmiennaReferencyjna := ADR(wTemperaturaZasilania_Lo);
	intPetlaPierwszySkan := intPetlaPierwszySkan + 1;
	
	arModbusOdczytCykliczny[intPetlaPierwszySkan].bAdresUrzadzenia := bAdres;
	arModbusOdczytCykliczny[intPetlaPierwszySkan].bFunkcja := TO_BYTE(enumModbusKodyFunkcji.OdczytNRejestrow);
	arModbusOdczytCykliczny[intPetlaPierwszySkan].uiAdresRejestru := 266;
	arModbusOdczytCykliczny[intPetlaPierwszySkan].ltCzestotliwosc := TIME_TO_LTIME(tMinimalnyCzasRaportowania);
	arModbusOdczytCykliczny[intPetlaPierwszySkan].pZmiennaReferencyjna := ADR(wTemperaturaPowrotu_Hi);
	intPetlaPierwszySkan := intPetlaPierwszySkan + 1;	
	
	arModbusOdczytCykliczny[intPetlaPierwszySkan].bAdresUrzadzenia := bAdres;
	arModbusOdczytCykliczny[intPetlaPierwszySkan].bFunkcja := TO_BYTE(enumModbusKodyFunkcji.OdczytNRejestrow);
	arModbusOdczytCykliczny[intPetlaPierwszySkan].uiAdresRejestru := 267;
	arModbusOdczytCykliczny[intPetlaPierwszySkan].ltCzestotliwosc := TIME_TO_LTIME(tMinimalnyCzasRaportowania);
	arModbusOdczytCykliczny[intPetlaPierwszySkan].pZmiennaReferencyjna := ADR(wTemperaturaPowrotu_Lo);
	intPetlaPierwszySkan := intPetlaPierwszySkan + 1;
		
	arModbusOdczytCykliczny[intPetlaPierwszySkan].bAdresUrzadzenia := bAdres;
	arModbusOdczytCykliczny[intPetlaPierwszySkan].bFunkcja := TO_BYTE(enumModbusKodyFunkcji.OdczytNRejestrow);
	arModbusOdczytCykliczny[intPetlaPierwszySkan].uiAdresRejestru := 272;
	arModbusOdczytCykliczny[intPetlaPierwszySkan].ltCzestotliwosc := TIME_TO_LTIME(tMinimalnyCzasRaportowania);
	arModbusOdczytCykliczny[intPetlaPierwszySkan].pZmiennaReferencyjna := ADR(wEnergiaCieplnaJednostka);
	intPetlaPierwszySkan := intPetlaPierwszySkan + 1;
	
	arModbusOdczytCykliczny[intPetlaPierwszySkan].bAdresUrzadzenia := bAdres;
	arModbusOdczytCykliczny[intPetlaPierwszySkan].bFunkcja := TO_BYTE(enumModbusKodyFunkcji.OdczytNRejestrow);
	arModbusOdczytCykliczny[intPetlaPierwszySkan].uiAdresRejestru := 273;
	arModbusOdczytCykliczny[intPetlaPierwszySkan].ltCzestotliwosc := TIME_TO_LTIME(tMinimalnyCzasRaportowania);
	arModbusOdczytCykliczny[intPetlaPierwszySkan].pZmiennaReferencyjna := ADR(wPrzeplywJednostka);
	intPetlaPierwszySkan := intPetlaPierwszySkan + 1;
	
	arModbusOdczytCykliczny[intPetlaPierwszySkan].bAdresUrzadzenia := bAdres;
	arModbusOdczytCykliczny[intPetlaPierwszySkan].bFunkcja := TO_BYTE(enumModbusKodyFunkcji.OdczytNRejestrow);
	arModbusOdczytCykliczny[intPetlaPierwszySkan].uiAdresRejestru := 274;
	arModbusOdczytCykliczny[intPetlaPierwszySkan].ltCzestotliwosc := TIME_TO_LTIME(tMinimalnyCzasRaportowania);
	arModbusOdczytCykliczny[intPetlaPierwszySkan].pZmiennaReferencyjna := ADR(wObjetoscJednostka);
	intPetlaPierwszySkan := intPetlaPierwszySkan + 1;
	
	arModbusOdczytCykliczny[intPetlaPierwszySkan].bAdresUrzadzenia := bAdres;
	arModbusOdczytCykliczny[intPetlaPierwszySkan].bFunkcja := TO_BYTE(enumModbusKodyFunkcji.OdczytNRejestrow);
	arModbusOdczytCykliczny[intPetlaPierwszySkan].uiAdresRejestru := 275;
	arModbusOdczytCykliczny[intPetlaPierwszySkan].ltCzestotliwosc := TIME_TO_LTIME(tMinimalnyCzasRaportowania);
	arModbusOdczytCykliczny[intPetlaPierwszySkan].pZmiennaReferencyjna := ADR(wMocJednostka);
	intPetlaPierwszySkan := intPetlaPierwszySkan + 1;
END_IF

// konwersja 2 odczytanych wordów na 32Float
fnKonwersja2x16naFloat32BySchneider(wRejestrMSW := wEnergiaCieplna_Hi, wRejestrLSW := wEnergiaCieplna_Lo, rWartoscFloat32 := rEnergiaCieplna);
fnKonwersja2x16naFloat32BySchneider(wRejestrMSW := wPrzeplyw_Hi, wRejestrLSW := wPrzeplyw_Lo, rWartoscFloat32 := rPrzeplyw);
fnKonwersja2x16naFloat32BySchneider(wRejestrMSW := wObjetosc_Hi, wRejestrLSW := wObjetosc_Lo, rWartoscFloat32 := rObjetosc);
fnKonwersja2x16naFloat32BySchneider(wRejestrMSW := wMoc_Hi, wRejestrLSW := wMoc_Lo, rWartoscFloat32 := rMoc);
fnKonwersja2x16naFloat32BySchneider(wRejestrMSW := wTemperaturaZasilania_Hi, wRejestrLSW := wTemperaturaZasilania_Lo, rWartoscFloat32 := rTemperaturaZasilania);
fnKonwersja2x16naFloat32BySchneider(wRejestrMSW := wTemperaturaPowrotu_Hi, wRejestrLSW := wTemperaturaPowrotu_Lo, rWartoscFloat32 := rTemperaturaPowrotu);

// Przeliczenie zmiennych
fbEnergiaCieplna(	rWartoscWejsciowa := rEnergiaCieplna,
					rDeadband := 100,
					tCzasMinimalny := tMinimalnyCzasRaportowania,
					tCzasMaksymalny := tMaksymalnyCzasRaportowania,
					rWynikMnoznik := 1000000000,
					rWynikOffset := 0,
					rWartoscWejsciowaZaraportowana := rEnergiaCieplnaZaraportowana,
					rWartoscWyjsciowa => rEnergiaCieplna);
					
fbPrzeplyw(	rWartoscWejsciowa := rPrzeplyw,
			rDeadband := 0.00000027778,
			tCzasMinimalny := tMinimalnyCzasRaportowania,
			tCzasMaksymalny := tMaksymalnyCzasRaportowania,
			rWynikMnoznik := 0.00000027778,
			rWynikOffset := 0,
			rWartoscWejsciowaZaraportowana := rPrzeplywZaraportowana,
			rWartoscWyjsciowa => rPrzeplyw);
							
fbObjetosc(	rWartoscWejsciowa := rObjetosc,
			rDeadband := 0.001,
			tCzasMinimalny := tMinimalnyCzasRaportowania,
			tCzasMaksymalny := tMaksymalnyCzasRaportowania,
			rWynikMnoznik := 1,
			rWynikOffset := 0,
			rWartoscWejsciowaZaraportowana := rObjetoscZaraportowana,
			rWartoscWyjsciowa => rObjetosc);								
								
fbMoc(	rWartoscWejsciowa := rMoc,
		rDeadband := 10,
		tCzasMinimalny := tMinimalnyCzasRaportowania,
		tCzasMaksymalny := tMaksymalnyCzasRaportowania,
		rWynikMnoznik := 1000,
		rWynikOffset := 0,
		rWartoscWejsciowaZaraportowana := rMocZaraportowana,
		rWartoscWyjsciowa => rMoc);
				
fbTemperaturaZasilania(	rWartoscWejsciowa := rTemperaturaZasilania,
						rDeadband := 0.1,
						tCzasMinimalny := tMinimalnyCzasRaportowania,
						tCzasMaksymalny := tMaksymalnyCzasRaportowania,
						rWynikMnoznik := 1,
						rWynikOffset := 273.15,
						rWartoscWejsciowaZaraportowana := rTemperaturaZasilaniaZaraportowana,
						rWartoscWyjsciowa => rTemperaturaZasilania);
			
fbTemperaturaPowrotu(	rWartoscWejsciowa := rTemperaturaPowrotu,
						rDeadband := 0.1,
						tCzasMinimalny := tMinimalnyCzasRaportowania,
						tCzasMaksymalny := tMaksymalnyCzasRaportowania,
						rWynikMnoznik := 1,
						rWynikOffset := 273.15,
						rWartoscWejsciowaZaraportowana := rTemperaturaPowrotuZaraportowana,
						rWartoscWyjsciowa => rTemperaturaPowrotu);							

// Sprawdzanie czy pomiar aktualnego przeplywu działa (alarm jest generowany, jeśli odczyt nie zmienił wartości w przeciągu 12h)
IF rPrzeplywPamiec = rPrzeplyw THEN
	xBrakZmianyPrzeplywu := TRUE;
ELSE
	xBrakZmianyPrzeplywu := FALSE;	
END_IF
fbBrakZmianyPrzeplywuTimer(IN := xBrakZmianyPrzeplywu, PT := T#12H);
IF fbBrakZmianyPrzeplywuTimer.Q THEN
	xBladBrakZmianyPrzeplywu := TRUE;
ELSE
	xBladBrakZmianyPrzeplywu := FALSE;
END_IF
rPrzeplywPamiec := rPrzeplyw;

// Sprawdzanie czy pomiar temperatury zasilania działa (alarm jest generowany, jeśli odczyt nie zmienił wartości w przeciągu 12h)
IF rTemperaturaZasilaniaPamiec = rTemperaturaZasilania THEN
	xBrakZmianyTemperaturyZasilania := TRUE;
ELSE
	xBrakZmianyTemperaturyZasilania := FALSE;	
END_IF
fbBrakZmianyTemperaturyZasilaniaTimer(IN := xBrakZmianyTemperaturyZasilania, PT := T#12H);
IF fbBrakZmianyTemperaturyZasilaniaTimer.Q THEN
	xBladBrakZmianyTemperaturyZasilania := TRUE;
ELSE
	xBladBrakZmianyTemperaturyZasilania := FALSE;
END_IF
rTemperaturaZasilaniaPamiec := rTemperaturaZasilania;

// Sprawdzanie czy pomiar temperatury powrotu działa (alarm jest generowany, jeśli odczyt nie zmienił wartości w przeciągu 12h)
IF rTemperaturaPowrotuPamiec = rTemperaturaPowrotu THEN
	xBrakZmianyTemperaturyPowrotu := TRUE;
ELSE
	xBrakZmianyTemperaturyPowrotu := FALSE;	
END_IF
fbBrakZmianyTemperaturyPowrotuTimer(IN := xBrakZmianyTemperaturyPowrotu, PT := T#12H);
IF fbBrakZmianyTemperaturyPowrotuTimer.Q THEN
	xBladBrakZmianyTemperaturyPowrotu := TRUE;
ELSE
	xBladBrakZmianyTemperaturyPowrotu := FALSE;
END_IF
rTemperaturaPowrotuPamiec := rTemperaturaPowrotu;

// Obsluga komunikatu przychodzacego z IZE
IF sKomunikat <> sKomunikatPamiec AND xPoInicjalizacji THEN
	sKomunikatPamiec := sKomunikat;
	IF fnIDOdbiorcyMatch(sKomunikat , sIdInstancji) THEN
		sDane := '';
		//zapytanie typu Q
		IF fnKomunikatTyp(sKomunikat) = 'Q' AND arModbusStatusKomunikacji[bAdres] = enumModbusStatus.KomunikacjaPrawidlowa THEN
			IF fnKomunikatDaneSzukajWartosci(sKomunikat , 'ENCC=') = '?' OR fnKomunikatDaneSzukajWartosci(sKomunikat , 'ALL=') = '?' THEN
				fnKomunikatDaneDodaj_xOverFlow(sDane := sDane , sAtrybut := 'ENCC=' , sWartosc := REAL_TO_STRING(rEnergiaCieplna) , xOverFlow := xOverFlow);	
				IF xOverFlow = TRUE THEN
					fnZapiszKomunikat(	sCalyKomunikat := '' ,
										sTypKomunikatu := 'A' ,
										sMnemonik := sMnemonik ,
										sMACAdres := sMACAdres ,
										sIDNadawcy := sIdInstancji ,
										sIDOdbiorcy := sIdAplikacji ,
										sDaneZapasowe := sDaneZapasowe ,
										sDane := sDane ,
										arTablicaKomunikatow := arTablicaKomunikatow ,
										intTablicaKomunikatowZnacznikZapisu := intTablicaKomunikatowZnacznikZapisu ,
										intTablicaKomunikatowRozmiar := intTablicaKomunikatowRozmiar ,
										sWyslanyKomunikat := sWyslanyKomunikatDummy);
					sDane := '';
				END_IF
			END_IF
			IF fnKomunikatDaneSzukajWartosci(sKomunikat , 'FLOWCC=') = '?' OR fnKomunikatDaneSzukajWartosci(sKomunikat , 'ALL=') = '?' THEN
				fnKomunikatDaneDodaj_xOverFlow(sDane := sDane , sAtrybut := 'FLOWCC=' , sWartosc := REAL_TO_STRING(rPrzeplyw) , xOverFlow := xOverFlow);	
				IF xOverFlow = TRUE THEN
					fnZapiszKomunikat(	sCalyKomunikat := '' ,
										sTypKomunikatu := 'A' ,
										sMnemonik := sMnemonik ,
										sMACAdres := sMACAdres ,
										sIDNadawcy := sIdInstancji ,
										sIDOdbiorcy := sIdAplikacji ,
										sDaneZapasowe := sDaneZapasowe ,
										sDane := sDane ,
										arTablicaKomunikatow := arTablicaKomunikatow ,
										intTablicaKomunikatowZnacznikZapisu := intTablicaKomunikatowZnacznikZapisu ,
										intTablicaKomunikatowRozmiar := intTablicaKomunikatowRozmiar ,
										sWyslanyKomunikat := sWyslanyKomunikatDummy);
					sDane := '';
				END_IF
			END_IF
			IF fnKomunikatDaneSzukajWartosci(sKomunikat , 'VOLCC=') = '?' OR fnKomunikatDaneSzukajWartosci(sKomunikat , 'ALL=') = '?' THEN
				fnKomunikatDaneDodaj_xOverFlow(sDane := sDane , sAtrybut := 'VOLCC=' , sWartosc := REAL_TO_STRING(rObjetosc) , xOverFlow := xOverFlow);	
				IF xOverFlow = TRUE THEN
					fnZapiszKomunikat(	sCalyKomunikat := '' ,
										sTypKomunikatu := 'A' ,
										sMnemonik := sMnemonik ,
										sMACAdres := sMACAdres ,
										sIDNadawcy := sIdInstancji ,
										sIDOdbiorcy := sIdAplikacji ,
										sDaneZapasowe := sDaneZapasowe ,
										sDane := sDane ,
										arTablicaKomunikatow := arTablicaKomunikatow ,
										intTablicaKomunikatowZnacznikZapisu := intTablicaKomunikatowZnacznikZapisu ,
										intTablicaKomunikatowRozmiar := intTablicaKomunikatowRozmiar ,
										sWyslanyKomunikat := sWyslanyKomunikatDummy);
					sDane := '';
				END_IF
			END_IF
			IF fnKomunikatDaneSzukajWartosci(sKomunikat , 'POWCC=') = '?' OR fnKomunikatDaneSzukajWartosci(sKomunikat , 'ALL=') = '?' THEN
				fnKomunikatDaneDodaj_xOverFlow(sDane := sDane , sAtrybut := 'POWCC=' , sWartosc := REAL_TO_STRING(rMoc) , xOverFlow := xOverFlow);	
				IF xOverFlow = TRUE THEN
					fnZapiszKomunikat(	sCalyKomunikat := '' ,
										sTypKomunikatu := 'A' ,
										sMnemonik := sMnemonik ,
										sMACAdres := sMACAdres ,
										sIDNadawcy := sIdInstancji ,
										sIDOdbiorcy := sIdAplikacji ,
										sDaneZapasowe := sDaneZapasowe ,
										sDane := sDane ,
										arTablicaKomunikatow := arTablicaKomunikatow ,
										intTablicaKomunikatowZnacznikZapisu := intTablicaKomunikatowZnacznikZapisu ,
										intTablicaKomunikatowRozmiar := intTablicaKomunikatowRozmiar ,
										sWyslanyKomunikat := sWyslanyKomunikatDummy);
					sDane := '';
				END_IF
			END_IF
			IF fnKomunikatDaneSzukajWartosci(sKomunikat , 'TEMPINCC=') = '?' OR fnKomunikatDaneSzukajWartosci(sKomunikat , 'ALL=') = '?' THEN
				fnKomunikatDaneDodaj_xOverFlow(sDane := sDane , sAtrybut := 'TEMPINCC=' , sWartosc := REAL_TO_STRING(rTemperaturaZasilania) , xOverFlow := xOverFlow);	
				IF xOverFlow = TRUE THEN
					fnZapiszKomunikat(	sCalyKomunikat := '' ,
										sTypKomunikatu := 'A' ,
										sMnemonik := sMnemonik ,
										sMACAdres := sMACAdres ,
										sIDNadawcy := sIdInstancji ,
										sIDOdbiorcy := sIdAplikacji ,
										sDaneZapasowe := sDaneZapasowe ,
										sDane := sDane ,
										arTablicaKomunikatow := arTablicaKomunikatow ,
										intTablicaKomunikatowZnacznikZapisu := intTablicaKomunikatowZnacznikZapisu ,
										intTablicaKomunikatowRozmiar := intTablicaKomunikatowRozmiar ,
										sWyslanyKomunikat := sWyslanyKomunikatDummy);
					sDane := '';
				END_IF
			END_IF
			IF fnKomunikatDaneSzukajWartosci(sKomunikat , 'TEMPOUTCC=') = '?' OR fnKomunikatDaneSzukajWartosci(sKomunikat , 'ALL=') = '?' THEN
				fnKomunikatDaneDodaj_xOverFlow(sDane := sDane , sAtrybut := 'TEMPOUTCC=' , sWartosc := REAL_TO_STRING(rTemperaturaPowrotu) , xOverFlow := xOverFlow);	
				IF xOverFlow = TRUE THEN
					fnZapiszKomunikat(	sCalyKomunikat := '' ,
										sTypKomunikatu := 'A' ,
										sMnemonik := sMnemonik ,
										sMACAdres := sMACAdres ,
										sIDNadawcy := sIdInstancji ,
										sIDOdbiorcy := sIdAplikacji ,
										sDaneZapasowe := sDaneZapasowe ,
										sDane := sDane ,
										arTablicaKomunikatow := arTablicaKomunikatow ,
										intTablicaKomunikatowZnacznikZapisu := intTablicaKomunikatowZnacznikZapisu ,
										intTablicaKomunikatowRozmiar := intTablicaKomunikatowRozmiar ,
										sWyslanyKomunikat := sWyslanyKomunikatDummy);
					sDane := '';
				END_IF
			END_IF
			// Pytanie o stany alarmów
			IF fnKomunikatDaneSzukajWartosci(sKomunikat , 'ALARM=') = '?' OR fnKomunikatDaneSzukajWartosci(sKomunikat , 'ALL=') = '?' THEN
				FOR intPetla := 1 TO 10 BY 1 DO
					// Raportowanie typu E (stanów alarmów) na zapytanie typu Q
					IF arErrorStan[intPetla] <> enumAlarmWartosc.StanNieznany THEN
						fnZapiszKomunikat(	sCalyKomunikat := '' ,
											sTypKomunikatu := 'E' ,
											sMnemonik := sMnemonik ,
											sMACAdres := sMACAdres ,
											sIDNadawcy := sIdInstancji ,
											sIDOdbiorcy := sIdAplikacji ,
											sDaneZapasowe := sDaneZapasowe ,
											sDane := fnKomunikatDaneErrorRetry(xAktywny := arErrorStan[intPetla] = enumAlarmWartosc.StanAlarmowy , intKlasa := arErrorKlasa[intPetla] , intNumer := intPetla),
											arTablicaKomunikatow := arTablicaKomunikatow ,
											intTablicaKomunikatowZnacznikZapisu := intTablicaKomunikatowZnacznikZapisu ,
											intTablicaKomunikatowRozmiar := intTablicaKomunikatowRozmiar ,
											sWyslanyKomunikat := sWyslanyKomunikatDummy);
					END_IF
				END_FOR
			END_IF
		END_IF
		// Raportowanie typu A na zapytanie Q
		IF sDane <> '' THEN
			fnZapiszKomunikat(	sCalyKomunikat := '' ,
								sTypKomunikatu := 'A' ,
								sMnemonik := sMnemonik ,
								sMACAdres := sMACAdres ,
								sIDNadawcy := sIdInstancji ,
								sIDOdbiorcy := sIdAplikacji ,
								sDaneZapasowe := sDaneZapasowe ,
								sDane := sDane ,
								arTablicaKomunikatow := arTablicaKomunikatow ,
								intTablicaKomunikatowZnacznikZapisu := intTablicaKomunikatowZnacznikZapisu ,
								intTablicaKomunikatowRozmiar := intTablicaKomunikatowRozmiar ,
								sWyslanyKomunikat := sWyslanyKomunikatDummy);
		END_IF
	END_IF
END_IF

// Raportowanie typu M do IZE wartosci odczytanych z Modbusa	
IF 	(rPrzeplyw <> rPrzeplywZaraportowana OR rMoc <> rMocZaraportowana OR rEnergiaCieplna <> rEnergiaCieplnaZaraportowana OR rObjetosc <> rObjetoscZaraportowana OR 
	rTemperaturaZasilania <> rTemperaturaZasilaniaZaraportowana OR rTemperaturaPowrotu <> rTemperaturaPowrotuZaraportowana) AND 
	arModbusStatusKomunikacji[bAdres] = enumModbusStatus.KomunikacjaPrawidlowa AND xPoInicjalizacji THEN
	xRaport := TRUE;
END_IF

